// TIA Portal V20 program export: 7 tag tables, 9 data types, 119 data blocks, 46 code blocks (in call order from the OBs), 106 instance data blocks

VAR_GLOBAL   // PLC tag table "00_Simulation"
END_VAR

VAR_GLOBAL   // PLC tag table "06_ProductionData"
END_VAR
VAR_GLOBAL CONSTANT   // user constants
   NO_DATASETS_CYCLETIMER : Int := 14;   // SICAR: Number of data sets Cycle Timer
   NO_DATASETS_LIMITVALUES : Int := 2;   // SICAR: Number of data sets Limit Value
   NO_DATASETS_SHIFTCOUNTER : Int := 2;   // SICAR: Number of data sets Shift Counter
   NO_DATASETS_COUNTER : Int := 2;   // SICAR: Number of data sets Counter
END_VAR

VAR_GLOBAL   // PLC tag table "07_Energy"
   "Active energy export tariff 1(F)" AT %ID624 : Real;
   "Active energy import tariff 1(F)" AT %ID612 : Real;
   "Active power L1" AT %ID644 : Real;
   "Active power L2" AT %ID648 : Real;
   "Active power L3" AT %ID652 : Real;
   "Apparent energy tariff 1 (F)" AT %ID620 : Real;
   "Apparent power L1" AT %ID632 : Real;
   "Apparent power L2" AT %ID636 : Real;
   "Apparent power L3" AT %ID640 : Real;
   PAC3220InPut AT %I500.0 : "LER_typePAC3220Input_Status";
   "Reactive energy export tariff 1 (F)" AT %ID628 : Real;
   "Reactive energy import tariff 1 (F)" AT %ID616 : Real;
   "Reactive power L1" AT %ID656 : Real;
   "Reactive power L2" AT %ID660 : Real;
   "Reactive power L3" AT %ID664 : Real;
   PAC3220OutPut AT %Q500.0 : "LER_typePAC3220Output_Status";
END_VAR
VAR_GLOBAL CONSTANT   // user constants
   NO_OF_MACHINES : USInt := 1;   // SICAR: No of machines for EE-Monitor
   NO_OF_MEASUREPOINTS : USInt := 10;   // SICAR: No of measurepoints for EE-Monitor
   "DP_FRWA1_1_0_000CC1-KE50~DP_FRWA1_1_0_000CC1-KE50_900" : Hw_Io := 10;
END_VAR

VAR_GLOBAL   // PLC tag table "08_CmInfo"
END_VAR
VAR_GLOBAL CONSTANT   // user constants
   NO_OF_RF_IDENT_DEVICES : USInt := 1;   // SICAR: Number of RF readers
   NO_OF_MV_IDENT_DEVICES : USInt := 1;   // SICAR: Number of MV readers
   NO_OF_ET200SPMOTORSTARTER : USInt := 1;   // SICAR: Number of ET200SP Motorstarter
END_VAR

VAR_GLOBAL   // PLC tag table "11_Settings"
END_VAR
VAR_GLOBAL CONSTANT   // user constants
   MAX_NO_OF_DEVICES_X1 : Int := 200;
   MAX_NO_OF_MODULES_X1 : Int := 200;
   MAX_NO_OF_DEVICES_X2 : Int := 200;
   MAX_NO_OF_MODULES_X2 : Int := 200;
END_VAR

VAR_GLOBAL   // PLC tag table "CentralFunctions"
END_VAR

VAR_GLOBAL   // PLC tag table "TextListId"
END_VAR
VAR_GLOBAL CONSTANT   // user constants
   TEXT_LIST_ID_PN_DEV_DIAG : Int := 591;   // SICAR: ID of PLC Alarm text list
   TEXT_LIST_ID_CHECKSUM : Int := 584;   // SICAR: ID of PLC Alarm text list
   TEXT_LIST_ID_EEEMONITOR_REPORT : Int := 562;   // SICAR: ID of PLC Alarm text list
   TEXT_LIST_ID_EEEMONITOR_CALC : Int := 561;   // SICAR: ID of PLC Alarm text list
   TEXT_LIST_ID_IDENT_SYSTEM : Int := 516;   // SICAR: ID of PLC Alarm for ident demo
   TEXT_LIST_ID_SMC_PD : Int := 585;   // SICAR: ID of PLC Alarm text list
   TEXT_LIST_ID_MOTORSTARTERS : Int := 588;   // SICAR: ID of PLC Alarm for motorstarter Demo
   TEXT_LIST_ID_DEV_FWD_REV : Int := 592;   // SICAR: ID of PLC Alarm for motorstarter Demo
END_VAR

TYPE "typeInspectionToStack"
   STRUCT
      partOn : Bool;
      signal1 : Bool;
      signal2 : Bool;
      signal3 : Bool;
      signal4 : Bool;
      signal5 : Bool;
      signal6 : Bool;
      signal7 : Bool;
      signal8 : Bool;
      signal9 : Bool;
      signal10 : Bool;
      signal11 : Bool;
      signal12 : Bool;
      signal13 : Bool;
      signal14 : Bool;
      signal15 : Bool;
      readyForOperation : Bool;
      signal17 : Bool;
      signal18 : Bool;
      signal19 : Bool;
      signal20 : Bool;
      signal21 : Bool;
      signal22 : Bool;
      signal23 : Bool;
      signal24 : Bool;
      signal25 : Bool;
      signal26 : Bool;
      signal27 : Bool;
      signal28 : Bool;
      signal29 : Bool;
      signal30 : Bool;
      signal31 : Bool;
      noInterference : Bool;
      collisionAreaOn : Bool;
      collisionAreaOff : Bool;
      girpped : Bool;
      unGirpped : Bool;
      signal37 : Bool;
      signal38 : Bool;
      signal39 : Bool;
      signal40 : Bool;
      signal41 : Bool;
      signal42 : Bool;
      signal43 : Bool;
      signal44 : Bool;
      signal45 : Bool;
      signal46 : Bool;
      signal47 : Bool;
      loadEnable : Bool;
      unGripRequest : Bool;
      loadComplete : Bool;
      signal51 : Bool;
      signal52 : Bool;
      signal53 : Bool;
      signal54 : Bool;
      signal55 : Bool;
      signal56 : Bool;
      signal57 : Bool;
      signal58 : Bool;
      signal59 : Bool;
      signal60 : Bool;
      signal61 : Bool;
      signal62 : Bool;
      signal63 : Bool;
      signal64 : Bool;
      signal65 : Bool;
      signal66 : Bool;
      signal67 : Bool;
      signal68 : Bool;
      signal69 : Bool;
      signal70 : Bool;
      signal71 : Bool;
      signal72 : Bool;
      signal73 : Bool;
      signal74 : Bool;
      signal75 : Bool;
      signal76 : Bool;
      signal77 : Bool;
      signal78 : Bool;
      signal79 : Bool;
      signal80 : Bool;
      signal81 : Bool;
      signal82 : Bool;
      signal83 : Bool;
      signal84 : Bool;
      signal85 : Bool;
      signal86 : Bool;
      signal87 : Bool;
      signal88 : Bool;
      signal89 : Bool;
      signal90 : Bool;
      signal91 : Bool;
      signal92 : Bool;
      signal93 : Bool;
      signal94 : Bool;
      signal95 : Bool;
   END_STRUCT;
END_TYPE

TYPE "typeStackToInspection"
   STRUCT
      partOn : Bool;
      signal1 : Bool;
      signal2 : Bool;
      signal3 : Bool;
      signal4 : Bool;
      signal5 : Bool;
      signal6 : Bool;
      signal7 : Bool;
      signal8 : Bool;
      signal9 : Bool;
      signal10 : Bool;
      signal11 : Bool;
      signal12 : Bool;
      signal13 : Bool;
      signal14 : Bool;
      signal15 : Bool;
      readyForOperation : Bool;
      signal17 : Bool;
      signal18 : Bool;
      signal19 : Bool;
      signal20 : Bool;
      signal21 : Bool;
      signal22 : Bool;
      signal23 : Bool;
      signal24 : Bool;
      signal25 : Bool;
      signal26 : Bool;
      signal27 : Bool;
      signal28 : Bool;
      signal29 : Bool;
      signal30 : Bool;
      signal31 : Bool;
      noInterference : Bool;
      collisionAreaOn : Bool;
      collisionAreaOff : Bool;
      girpped : Bool;
      unGirpped : Bool;
      signal37 : Bool;
      signal38 : Bool;
      signal39 : Bool;
      signal40 : Bool;
      signal41 : Bool;
      signal42 : Bool;
      signal43 : Bool;
      signal44 : Bool;
      signal45 : Bool;
      signal46 : Bool;
      signal47 : Bool;
      unloadRequest : Bool;
      gripRequest : Bool;
      unLoadComplete : Bool;
      signal51 : Bool;
      signal52 : Bool;
      signal53 : Bool;
      signal54 : Bool;
      signal55 : Bool;
      signal56 : Bool;
      signal57 : Bool;
      signal58 : Bool;
      signal59 : Bool;
      signal60 : Bool;
      signal61 : Bool;
      signal62 : Bool;
      signal63 : Bool;
      signal64 : Bool;
      signal65 : Bool;
      signal66 : Bool;
      signal67 : Bool;
      signal68 : Bool;
      signal69 : Bool;
      signal70 : Bool;
      signal71 : Bool;
      signal72 : Bool;
      signal73 : Bool;
      signal74 : Bool;
      signal75 : Bool;
      signal76 : Bool;
      signal77 : Bool;
      signal78 : Bool;
      signal79 : Bool;
      signal80 : Bool;
      signal81 : Bool;
      signal82 : Bool;
      signal83 : Bool;
      signal84 : Bool;
      signal85 : Bool;
      signal86 : Bool;
      signal87 : Bool;
      signal88 : Bool;
      signal89 : Bool;
      signal90 : Bool;
      signal91 : Bool;
      signal92 : Bool;
      signal93 : Bool;
      signal94 : Bool;
      signal95 : Bool;
   END_STRUCT;
END_TYPE

TYPE "typeEmMotorStarterInterface"
// stored: Access Published
   STRUCT
      EMmotorstarter : Array[0.."NO_OF_EM"] of "typeMotorStarterInterface";
   END_STRUCT;
END_TYPE

TYPE "typeEt200SpMotorstarterInterfaceHmi"
// stored: Access Published
   STRUCT
      et200SpMotorstarterReadValue : Bool;   // read Value of MotorStarter
      et200SpNumberOfMotorstarters { ExternalWritable := 'False'} : USInt;   // Number of Motor Starters
      et200SpUnitMotorstarter : USInt := 1;   // Unit selected
      et200SpEMMotorstarter : USInt := 0;   // Equipment Module selected
      et200SpMotorstarterCurrent : Array[0.."NO_OF_ET200SPMOTORSTARTER"] of Real;   // Current values
      et200SpMotorstarterInputs : Array[0.."NO_OF_ET200SPMOTORSTARTER"] of "LSicar_typeMotorstarterIn";   // Motorstarter Data Inputs HMI
      et200SpMotorstarterOutputs : Array[0.."NO_OF_ET200SPMOTORSTARTER"] of "LSicar_typeMotorstarterOut";   // Motorstarter Data Outputs HMI
   END_STRUCT;
END_TYPE

TYPE "typeMotorStarterInterface"
// stored: Access Published
   STRUCT
      et200SpMotorstarterCurrent : Array[0.."NO_OF_ET200SPMOTORSTARTER"] of Real;   // Current values
      et200SpMotorstarterInputs : Array[0.."NO_OF_ET200SPMOTORSTARTER"] of "LSicar_typeMotorstarterIn";   // Motorstarter Data Inputs HMI
      et200SpMotorstarterOutputs : Array[0.."NO_OF_ET200SPMOTORSTARTER"] of "LSicar_typeMotorstarterOut";   // Motorstarter Data Outputs HMI
   END_STRUCT;
END_TYPE

TYPE "typeEMIdentMv"
// stored: Access Published
   STRUCT
      identMvEM : Array[0.."NO_OF_EM"] of "typeIdentMvHmi";
   END_STRUCT;
END_TYPE

TYPE "typeIdentMvHmi"
// stored: Access Published
   STRUCT
      selectedUnit : USInt;
      selectedEM : USInt;
      mvReaderId : USInt;   // MV Reader ID
      numberOfMv : USInt;   // Number of used MV readers
      mvReader : Array[0.."NO_OF_MV_IDENT_DEVICES"] of "LSicar_typeIdentInterfaceHmi";   // MV Reader
   END_STRUCT;
END_TYPE

TYPE "typeEMIdentRf"
// stored: Access Published
   STRUCT
      identRfEM : Array[0.."NO_OF_EM"] of "typeIdentRfHmi";
   END_STRUCT;
END_TYPE

TYPE "typeIdentRfHmi"
// stored: Access Published
   STRUCT
      selectedUnit : USInt;
      selectedEM : USInt;
      rfReaderId : USInt;   // RF Reader ID
      numberOfRf : USInt;   // Number of used RFIDs
      rfReader : Array[0.."NO_OF_RF_IDENT_DEVICES"] of "LSicar_typeIdentInterfaceHmi";   // RF Reader
   END_STRUCT;
END_TYPE

DATA_BLOCK "Hmi"   // DB199
// stored: MemoryReserve 100
   VAR
      mainHeader : Array[0.."NO_OF_PANELS"] of "LAF_typeHeader";   // Input from the status bar of the HMI
      operationInterlock : "LAF_typeOperationInterlockInterface";
   END_VAR
BEGIN
   mainHeader[0].plcToHmi.modeRequestsButtons.operatorControlAllowed := 16#003F;
   mainHeader[1].plcToHmi.stateCommandsButtons.visibility := 16#F;
   mainHeader[1].plcToHmi.stateCommandsButtons.operatorControlAllowed := 16#F;
   mainHeader[0].plcToHmi.specialFunctionButtons.visibility := 16#00330F7307337077;
   mainHeader[0].plcToHmi.specialFunctionButtons.operatorControlAllowed := 16#00330F7307337077;
END_DATA_BLOCK

DATA_BLOCK "LRemoteAccess_Data"   // DB275
TITLE = Data
AUTHOR : Siemens
// Storing data about mobile panel and UCP connection status
// stored: MemoryReserve 100
   VAR
      mobilePanel1 : "LRemoteAccess_typeMobilePanel";
      connectionBoxes : Array[1..2] of "LRemoteAccess_typeConnectionBox";
      ActivationMobileDP { S7_SetPoint := 'True'} : "LRemoteAccess_typeMobile_DeActivate";   // Activate Mobile Panel
      DeactivationMobileDP { S7_SetPoint := 'True'} : "LRemoteAccess_typeMobile_DeActivate";   // Deactivate Mobile Panel
      connectionTimeout { S7_SetPoint := 'True'} : Time := T#5s;   // Connection timeout. Keep greater than 3 sec. Default 5 sec.
   END_VAR
BEGIN
   connectionBoxes[1].ID := 20;
   connectionBoxes[2].ID := 21;
END_DATA_BLOCK

DATA_BLOCK "Simulation"   // DB134
TITLE = Simulation
// Simulation data
// stored: MemoryReserve 100
   VAR
      data : "LAF_typeSimulation";
   END_VAR
BEGIN
   data.simulationActiveHmi := true;
END_DATA_BLOCK

DATA_BLOCK "HMI_Interface_Overview"   // DB276
// stored: Access Published, MemoryReserve 100
   VAR
      State : Struct
         "Anode Reel Cut" : "HMI_IF_OverView_Unit_UDT";
         "Cathode Reel Cut" : "HMI_IF_OverView_Unit_UDT";
         "Stacker #1" : "HMI_IF_OverView_Unit_UDT";
         "Stacker #2" : "HMI_IF_OverView_Unit_UDT";
         Inspection : "HMI_IF_OverView_Unit_UDT";
      END_STRUCT;
      homeCodition : Array[0..13] of "LER_typeEmOverviewHomeCondition";
   END_VAR
BEGIN
END_DATA_BLOCK

DATA_BLOCK "HMI_Interface_Parameter"   // DB262
// stored: Access Published, MemoryReserve 100
   VAR
      ProcessUnitSelect : Int := 5;   // 1. Anode Reel Cut, 2. Cathode Reel Cut, 3. Stacking#1, 4.Stacking#2, 5. Inspection
      Recipe : "HMI_IF_Parameter_LIstRecipe_Interface";
   END_VAR
   VAR RETAIN
      Parameter : Array[0..20] of "HMI_IF_Parameter_Parameter_UDT";
      Softcam : Array[0..23] of "LER_typeSoftCamRelation";
   END_VAR
   VAR
      RecipeButton : "HMI_IF_Parameter_Save Button_UDT";
      FATModeSelect : "LER_TypeFATMode_ModeSelect";
   END_VAR
   VAR RETAIN
      FATModeInterface : "LER_TypeFATModeInterface";
   END_VAR
   VAR
      teachingPosInterface { S7_SetPoint := 'True'} : Array[0..48] of "LER_TypeTeachingPosInterface";
      TeachingPos_Index { S7_SetPoint := 'True'} : SInt;
   END_VAR
BEGIN
END_DATA_BLOCK

DATA_BLOCK "RecipeParameter"   // DB168
// stored: MemoryReserve 100
   VAR
      unitRecipe : "LER_typeRecipe";
      ParameterSV { S7_SetPoint := 'True'} : "HMI_IF_Parameter_ListRecipe_UDT";
      ParameterPV { S7_SetPoint := 'True'} : "HMI_IF_Parameter_ListRecipe_UDT";
   END_VAR
BEGIN
   ParameterSV.Recipe6 := 9000000.0;
   ParameterSV.Recipe7 := 9000000.0;
   ParameterPV.Recipe6 := 300000.0;
   ParameterPV.Recipe7 := 300000.0;
END_DATA_BLOCK

DATA_BLOCK "LAF_InternalManual"   // DB43
VERSION : 19.0
// stored: MemoryReserve 100
   VAR
      hmi : Array[1..1] of "LAF_typeManHmiDisp";   // number of HMIs - modify the array size based on the required HMIs
      manualOperationEnabled : Bool;   // feedback whether the manual operation lines are selected
      emsWithManualOpConfigured { ExternalWritable := 'False'} : "LGM_emsWithManualOpConfigured";   // List of EMs with manual operation configured, for HMI button visibility
      disableUnit1 { S7_SetPoint := 'True'} : Bool;
      RisingEdge : Bool;
   END_VAR
BEGIN
END_DATA_BLOCK

DATA_BLOCK "ManualOperationControl_Template"   // DB197
// stored: MemoryReserve 100
   VAR
      manualOperationEm { ExternalAccessible := 'False'; ExternalVisible := 'False'; ExternalWritable := 'False'} : "LAF_typeManEm";
      manualOperationEmArea { ExternalAccessible := 'False'; ExternalVisible := 'False'; ExternalWritable := 'False'} : Array[1..1] of "LAF_typeManOperationArea";
      manualOperationCms { ExternalAccessible := 'False'; ExternalVisible := 'False'; ExternalWritable := 'False'} : Array[1..1] of "LAF_typeManOperation";
   END_VAR
BEGIN
   manualOperationEm.equipmentModuleNum := 3400;
END_DATA_BLOCK

DATA_BLOCK "HMI_Interface_DeviceHistory"   // DB7
// stored: MemoryReserve 100
   VAR
      hotPressLeftHistory { ExternalWritable := 'False'; S7_SetPoint := 'True'} : "LER_typeVisionInspectData";
      hotPressRightHistory { ExternalWritable := 'False'; S7_SetPoint := 'True'} : "LER_typeVisionInspectData";
      hipotHistory { ExternalWritable := 'False'; S7_SetPoint := 'True'} : "LER_typeHipotDataLog";
      thicknessHistory { ExternalWritable := 'False'; S7_SetPoint := 'True'} : "LER_typeThicknessDataLog";
      visionHistory { ExternalWritable := 'False'; S7_SetPoint := 'True'} : "LER_typeVisionHistory";
      laserMarkHistory { ExternalWritable := 'False'; S7_SetPoint := 'True'} : "LER_typeQRMarkerDataLog";
      weightCheckHistory { ExternalWritable := 'False'; S7_SetPoint := 'True'} : "LER_typeWeightCheckDataLog";
   END_VAR
BEGIN
END_DATA_BLOCK

DATA_BLOCK "OperatorPrompts"   // DB123
// stored: Access Published, MemoryReserve 100
   VAR
      triggers { ExternalAccessible := 'False'; ExternalVisible := 'False'; ExternalWritable := 'False'} : Array[1..63] of Bool;
      activeOperatorPrompt { ExternalWritable := 'False'} : Int;
      ack : Bool;
   END_VAR
BEGIN
END_DATA_BLOCK

DATA_BLOCK "ProdDataInterfaceHmi"   // DB53
TITLE = HMI and user interface for production data
AUTHOR : SICAR
FAMILY : ProdData
// DESCRIPTION OF FUNCTIONS:
// stored: MemoryReserve 100
   VAR RETAIN
      numberOfDataSets : "LSicar_typeNumberOfDataSets";   // Number of configured data sets
   END_VAR
   VAR
      colorCodeLimitSummary : UInt;   // Overall status Limit values
      colorCodeLimitSelButton : Array[0..8] of UInt;   // Color code for data set select button (Limit values)
   END_VAR
   VAR RETAIN
      limitValueDataSetSel : Int := 1;   // selected data set limit values
      limitDataSet : Array[0.."NO_DATASETS_LIMITVALUES"] of "LSicar_typeLimitValue";   // Data sets limit .values
      cycleTimerDataSetSel : Int := 1;   // selected data set cycle timer
      cycleTimerDataSet : Array[0.."NO_DATASETS_CYCLETIMER"] of "LSicar_typeCycleTimer";   // Data sets cycle timer
      counterDataSetSel : Int := 1;   // selected data set counter
      counterDataSet : Array[0.."NO_DATASETS_COUNTER"] of "LSicar_typeCounter";   // Data sets counter
      shiftCounterDataSetSel : Int := 1;   // selected data set shift counter
      shiftCounterDataSet : Array[0.."NO_DATASETS_SHIFTCOUNTER"] of "LSicar_typeShiftCounter";   // Data sets shift counter
      shiftCountOeeDataSetSel : Int := 1;   // selected data set OEE
      shiftCounterOeeDataSet : Array[0.."NO_DATASETS_SHIFTCOUNTER"] of "LSicar_typeShiftCounterOee";   // Data sets shift counter OEE
   END_VAR
BEGIN
END_DATA_BLOCK

DATA_BLOCK "ProdDataSimulation"   // DB5
{ DB_Accessible_From_OPC_UA := 'FALSE' }
// stored: DBAccessibleFromOPCUA false, DBAccessibleFromWebserver false, MemoryReserve 100
   VAR
      ProdDataCounter { ExternalAccessible := 'False'; ExternalVisible := 'False'; ExternalWritable := 'False'} : Struct   // Test tag prod data
         ProdDataCounter1Up1 : Bool;   // Test tag prod data
         ProdDataCounter1Up2 : Bool;   // Test tag prod data
         ProdDataCounter1Down1 : Bool;   // Test tag prod data
         ProdDataCounter1Down2 : Bool;   // Test tag prod data
         ProdDataCounter1Reset1 : Bool;   // Test tag prod data
         ProdDataCounter1Reset2 : Bool;   // Test tag prod data
         ProdDataCounter1ResetAll : Bool;   // Test tag prod data
         ProdDataCounter2Up1 : Bool;
         ProdDataCounter2Up2 : Bool;
         ProdDataCounter2Down1 : Bool;
         ProdDataCounter2Down2 : Bool;
         ProdDataCounter2Reset1 : Bool;
         ProdDataCounter2Reset2 : Bool;
         ProdDataCounter2ResetAll : Bool;
         userInterfaceVisibilityDataSet2Counter : DWord := 2#0000_0000_0000_0000_0000_0000_0000_0011;
         userInterfaceVisibilityDataSet1Counter : DWord := 2#0000_0000_0000_0000_0011_1111_1111_1111;
         ProdDataEnable : Bool;
      END_STRUCT;
      ProdDataCyclic { ExternalAccessible := 'False'; ExternalVisible := 'False'; ExternalWritable := 'False'} : Struct   // Test tag prod data
         cycleTimer1Run1 : Bool;   // Test tag prod data
         cycleTimer1Run2 : Bool;   // Test tag prod data
         cycleTimer1Hold1 : Bool;   // Test tag prod data
         cycleTimer1Hold2 : Bool;   // Test tag prod data
         cycleTimer1Reset1 : Bool;   // Test tag prod data
         cycleTimer1Reset2 : Bool;   // Test tag prod data
         cycleTimer1ResetAll : Bool;   // Test tag prod data
         cycleTimer2Run1 : Bool;   // Test tag prod data
         cycleTimer2Run2 : Bool;   // Test tag prod data
         cycleTimer2Hold1 : Bool;   // Test tag prod data
         cycleTimer2Hold2 : Bool;   // Test tag prod data
         cycleTimer2Reset1 : Bool;   // Test tag prod data
         cycleTimer2Reset2 : Bool;   // Test tag prod data
         cycleTimer2ResetAll : Bool;   // Test tag prod data
         cyclicTimerEnable : Bool;
         userInterfaceVisibilityDataSet1Cyclic : DWord := 2#0000_0000_0000_0000_0000_0000_0000_0111;
         userInterfaceVisibilityDataSet2Cyclic : DWord := 2#0000_0000_0000_0000_0000_0000_0000_0111;
         userInterfaceVisibilityDataSet3Cyclic : DWord := 2#0000_0000_0000_0000_0000_0000_1110_1111;
         userInterfaceVisibilityDataSet4Cyclic : DWord := 2#0000_0000_0000_0000_0011_1110_1111_1011;
         userInterfaceVisibilityDataSet5Cyclic : DWord := 2#0000_0000_0000_1111_1110_1111_1111_0111;
         userInterfaceVisibilityDataSet6Cyclic : DWord := 2#0000_0000_0000_0111_1111_1101_1111_1111;
         userInterfaceVisibilityDataSet7Cyclic : DWord := 2#0000_0000_0000_0000_0000_0000_0000_1111;
         userInterfaceVisibilityDataSet8Cyclic : DWord := 2#0000_0000_0000_0000_0000_0000_0000_1111;
         userInterfaceVisibilityDataSet9Cyclic : DWord := 2#0000_0000_0000_0000_0000_0000_0000_1111;
         userInterfaceVisibilityDataSet10Cyclic : DWord := 2#0000_0000_0000_0000_0000_0000_0000_1111;
         userInterfaceVisibilityDataSet11Cyclic : DWord := 2#0000_0000_0000_0000_0000_0000_0000_1111;
         userInterfaceVisibilityDataSet12Cyclic : DWord := 2#0000_0000_0000_0000_0000_0000_0000_1111;
         userInterfaceVisibilityDataSet13Cyclic : DWord := 2#0000_0000_0000_0000_0000_0000_0000_0111;
         userInterfaceVisibilityDataSet14Cyclic : DWord := 2#0000_0000_0000_0000_0000_0000_0000_1111;
      END_STRUCT;
      ProdDataLimitValues { ExternalAccessible := 'False'; ExternalVisible := 'False'; ExternalWritable := 'False'} : Struct   // Test tag prod data
         limitVal1Count1PreWarn1 : Bool;   // Test tag prod data
         limitVal1Count1PreWarn3 : Bool;   // Test tag prod data
         limitVal1Count1PreWarn2 : Bool;   // Test tag prod data
         limitVal1Count1Alarm1 : Bool;   // Test tag prod data
         limitVal1Count1Alarm3 : Bool;   // Test tag prod data
         limitVal1Count1Alarm2 : Bool;   // Test tag prod data
         limitVal1Count1 : Bool;   // Test tag prod data
         limitVal1Count2 : Bool;   // Test tag prod data
         limitVal1Count3 : Bool;   // Test tag prod data
         limitVal1Set1 : Bool;   // Test tag prod data
         limitVal1Set3 : Bool;   // Test tag prod data
         limitVal1Set2 : Bool;   // Test tag prod data
         limitValuesEnable : Bool;
         userInterfaceVisibilityDataSet2LimitValues : DWord := 2#0000_0000_0000_0000_0000_0011_1111_1111;
         userInterfaceVisibilityDataSet1LimitValues : DWord := 2#0000_0000_0000_0000_0000_0000_0000_1111;
      END_STRUCT;
      ProdDataShiftCounter { ExternalAccessible := 'False'; ExternalVisible := 'False'; ExternalWritable := 'False'} : Struct   // Test tag prod data
         shiftCounter1Cnt1Curr : Bool;   // Test tag prod data
         shiftCounter1Cnt1CurrOk : Bool;   // Test tag prod data
         shiftCounter1Cnt2Curr : Bool;   // Test tag prod data
         shiftCounter1Cnt2CurrOk : Bool;   // Test tag prod data
         shiftCounter1Cnt3Curr : Bool;   // Test tag prod data
         shiftCounter1Cnt3CurrOk : Bool;   // Test tag prod data
         shiftCounter1ResetAllExt : Bool;   // Test tag prod data
         ShiftCounterEnable : Bool;
         userInterfaceVisibilityDataSet2ShiftCounter : DWord := 2#0000_0000_0000_0000_0000_0011_1111_1111;
         userInterfaceVisibilityDataSet1ShiftCounter : DWord := 2#0000_0000_0000_0000_0000_0000_0000_1111;
      END_STRUCT;
      ProdDataShiftCounterOEE { ExternalAccessible := 'False'; ExternalVisible := 'False'; ExternalWritable := 'False'} : Struct   // Test tag prod data
         ShiftCounterOEEEnable : Bool;
         userInterfaceVisibilityDataSet2ShiftCounterOEE : DWord := 2#0000_0000_0000_0000_0000_0011_1111_1111;
         userInterfaceVisibilityDataSet1ShiftCounterOEE : DWord := 2#0000_0000_0000_0000_0000_0000_0000_1111;
      END_STRUCT;
   END_VAR
BEGIN
END_DATA_BLOCK

DATA_BLOCK "ShiftInitBools"   // DB257
// stored: MemoryReserve 100
   VAR
      earlyShift : Bool;
      lateShift : Bool;
      nightShift : Bool;
   END_VAR
BEGIN
END_DATA_BLOCK

DATA_BLOCK "ShiftTimesList"   // DB52
TITLE = Shift times
{ DB_Accessible_From_OPC_UA := 'FALSE' }
AUTHOR : SICAR
FAMILY : Shiftmodel
// Shift times List
// stored: DBAccessibleFromOPCUA false, MemoryReserve 100
   VAR
      list { ExternalAccessible := 'False'; ExternalVisible := 'False'; ExternalWritable := 'False'} : Array[0..10] of "LSicar_typeShiftmodTime1DaySel";   // Shiftmodel list
   END_VAR
BEGIN
   list[3].listValidFor.sunday := TRUE;
   list[4].listValidFor.sunday := FALSE;
   list[1..3].listValidFor.monday := TRUE;
   list[4].listValidFor.monday := FALSE;
   list[1..3].listValidFor.tuesday := TRUE;
   list[4].listValidFor.tuesday := FALSE;
   list[1..3].listValidFor.wednesday := TRUE;
   list[4].listValidFor.wednesday := FALSE;
   list[1..3].listValidFor.thursday := TRUE;
   list[4].listValidFor.thursday := FALSE;
   list[1].listValidFor.friday := TRUE;
   list[3].listValidFor.friday := TRUE;
   list[4].listValidFor.friday := FALSE;
   list[3].listValidFor.saturday := TRUE;
   list[4].listValidFor.saturday := FALSE;
   list[1].shift[1].endCircuitTime := TOD#05:57:00;
   list[1].shift[2].endCircuitTime := TOD#13:57:00;
   list[1].shift[3].endCircuitTime := TOD#21:57:00;
   list[2].shift[1].endCircuitTime := TOD#04:57:00;
   list[2].shift[2].endCircuitTime := TOD#14:27:00;
   list[3].shift[1].endCircuitTime := TOD#05:57:00;
   list[3].shift[2].endCircuitTime := TOD#14:27:00;
   list[3].shift[3].endCircuitTime := TOD#22:57:00;
   list[4].shift[1..3].endCircuitTime := TOD#00:00:00;
   list[1].shift[1].start := TOD#06:00:00;
   list[1].shift[2].start := TOD#14:00:00;
   list[1].shift[3].start := TOD#22:00:00;
   list[2].shift[1].start := TOD#05:00:00;
   list[2].shift[2].start := TOD#14:30:00;
   list[3].shift[1].start := TOD#06:00:00;
   list[3].shift[2].start := TOD#14:30:00;
   list[3].shift[3].start := TOD#23:00:00;
   list[4].shift[1..3].start := TOD#00:00:00;
   list[1].shift[1].break[1].start := TOD#08:00:00;
   list[1].shift[1].break[2].start := TOD#10:00:00;
   list[1].shift[1].break[3].start := TOD#12:00:00;
   list[1].shift[1].break[4].start := TOD#00:00:00;
   list[1].shift[2].break[1].start := TOD#16:00:00;
   list[1].shift[2].break[2].start := TOD#18:00:00;
   list[1].shift[2].break[3].start := TOD#20:00:00;
   list[1].shift[3].break[1].start := TOD#00:00:00;
   list[1].shift[3].break[2].start := TOD#02:00:00;
   list[1].shift[3].break[3].start := TOD#04:00:00;
   list[2].shift[1].break[1].start := TOD#07:00:00;
   list[2].shift[1].break[2].start := TOD#09:00:00;
   list[2].shift[1].break[3].start := TOD#11:00:00;
   list[2].shift[1].break[4].start := TOD#13:00:00;
   list[2].shift[2].break[1].start := TOD#16:30:00;
   list[2].shift[2].break[2].start := TOD#18:30:00;
   list[2].shift[2].break[3].start := TOD#20:30:00;
   list[2].shift[2].break[4].start := TOD#22:00:00;
   list[3].shift[1].break[1].start := TOD#08:00:00;
   list[3].shift[1].break[2].start := TOD#10:00:00;
   list[3].shift[1].break[3].start := TOD#11:30:00;
   list[3].shift[1].break[4].start := TOD#12:30:00;
   list[3].shift[2].break[1].start := TOD#16:00:00;
   list[3].shift[2].break[2].start := TOD#18:00:00;
   list[3].shift[2].break[3].start := TOD#19:30:00;
   list[3].shift[2].break[4].start := TOD#20:30:00;
   list[3].shift[3].break[1].start := TOD#00:00:00;
   list[3].shift[3].break[2].start := TOD#02:00:00;
   list[3].shift[3].break[3].start := TOD#03:30:00;
   list[3].shift[3].break[4].start := TOD#04:30:00;
   list[4].shift[1].break[1..4].start := TOD#00:00:00;
   list[4].shift[2].break[1..4].start := TOD#00:00:00;
   list[4].shift[3].break[1..4].start := TOD#00:00:00;
   list[1].shift[1].break[1].startCircuitTime := TOD#08:02:00;
   list[1].shift[1].break[2].startCircuitTime := TOD#00:00:00;
   list[1].shift[1].break[3].startCircuitTime := TOD#12:02:00;
   list[1].shift[1].break[4].startCircuitTime := TOD#00:00:00;
   list[1].shift[2].break[1].startCircuitTime := TOD#16:02:00;
   list[1].shift[2].break[2].startCircuitTime := TOD#00:00:00;
   list[1].shift[2].break[3].startCircuitTime := TOD#20:02:00;
   list[1].shift[3].break[1].startCircuitTime := TOD#00:02:00;
   list[1].shift[3].break[2].startCircuitTime := TOD#00:00:00;
   list[1].shift[3].break[3].startCircuitTime := TOD#04:02:00;
   list[2].shift[1].break[1].startCircuitTime := TOD#07:02:00;
   list[2].shift[1].break[2].startCircuitTime := TOD#00:00:00;
   list[2].shift[1].break[3].startCircuitTime := TOD#11:02:00;
   list[2].shift[1].break[4].startCircuitTime := TOD#13:02:00;
   list[2].shift[2].break[1].startCircuitTime := TOD#16:32:00;
   list[2].shift[2].break[2].startCircuitTime := TOD#00:00:00;
   list[2].shift[2].break[3].startCircuitTime := TOD#20:32:00;
   list[2].shift[2].break[4].startCircuitTime := TOD#22:02:00;
   list[3].shift[1].break[1].startCircuitTime := TOD#00:00:00;
   list[3].shift[1].break[2].startCircuitTime := TOD#10:02:00;
   list[3].shift[1].break[3].startCircuitTime := TOD#00:00:00;
   list[3].shift[1].break[4].startCircuitTime := TOD#12:32:00;
   list[3].shift[2].break[1].startCircuitTime := TOD#00:00:00;
   list[3].shift[2].break[2].startCircuitTime := TOD#18:02:00;
   list[3].shift[2].break[3].startCircuitTime := TOD#00:00:00;
   list[3].shift[2].break[4].startCircuitTime := TOD#20:32:00;
   list[3].shift[3].break[1].startCircuitTime := TOD#00:00:00;
   list[3].shift[3].break[2].startCircuitTime := TOD#02:02:00;
   list[3].shift[3].break[3..4].startCircuitTime := TOD#00:00:00;
   list[4].shift[1].break[1..4].startCircuitTime := TOD#00:00:00;
   list[4].shift[2].break[1..4].startCircuitTime := TOD#00:00:00;
   list[4].shift[3].break[1..4].startCircuitTime := TOD#00:00:00;
   list[1].shift[1].break[1].endCircuitTime := TOD#08:13:00;
   list[1].shift[1].break[2].endCircuitTime := TOD#00:00:00;
   list[1].shift[1].break[3].endCircuitTime := TOD#12:13:00;
   list[1].shift[1].break[4].endCircuitTime := TOD#00:00:00;
   list[1].shift[2].break[1].endCircuitTime := TOD#16:13:00;
   list[1].shift[2].break[2].endCircuitTime := TOD#00:00:00;
   list[1].shift[2].break[3].endCircuitTime := TOD#20:13:00;
   list[1].shift[3].break[1].endCircuitTime := TOD#00:13:00;
   list[1].shift[3].break[2].endCircuitTime := TOD#00:00:00;
   list[1].shift[3].break[3].endCircuitTime := TOD#04:13:00;
   list[2].shift[1].break[1].endCircuitTime := TOD#07:13:00;
   list[2].shift[1].break[2].endCircuitTime := TOD#00:00:00;
   list[2].shift[1].break[3].endCircuitTime := TOD#11:13:00;
   list[2].shift[1].break[4].endCircuitTime := TOD#13:13:00;
   list[2].shift[2].break[1].endCircuitTime := TOD#16:43:00;
   list[2].shift[2].break[2].endCircuitTime := TOD#00:00:00;
   list[2].shift[2].break[3].endCircuitTime := TOD#20:43:00;
   list[2].shift[2].break[4].endCircuitTime := TOD#22:13:00;
   list[3].shift[1].break[1].endCircuitTime := TOD#00:00:00;
   list[3].shift[1].break[2].endCircuitTime := TOD#10:13:00;
   list[3].shift[1].break[3].endCircuitTime := TOD#00:00:00;
   list[3].shift[1].break[4].endCircuitTime := TOD#12:43:00;
   list[3].shift[2].break[1].endCircuitTime := TOD#00:00:00;
   list[3].shift[2].break[2].endCircuitTime := TOD#18:13:00;
   list[3].shift[2].break[3].endCircuitTime := TOD#00:00:00;
   list[3].shift[2].break[4].endCircuitTime := TOD#20:43:00;
   list[3].shift[3].break[1].endCircuitTime := TOD#00:00:00;
   list[3].shift[3].break[2].endCircuitTime := TOD#02:13:00;
   list[3].shift[3].break[3..4].endCircuitTime := TOD#00:00:00;
   list[4].shift[1].break[1..4].endCircuitTime := TOD#00:00:00;
   list[4].shift[2].break[1..4].endCircuitTime := TOD#00:00:00;
   list[4].shift[3].break[1..4].endCircuitTime := TOD#00:00:00;
   list[1].shift[1].break[1].end := TOD#08:15:00;
   list[1].shift[1].break[2].end := TOD#10:10:00;
   list[1].shift[1].break[3].end := TOD#12:15:00;
   list[1].shift[1].break[4].end := TOD#00:00:00;
   list[1].shift[2].break[1].end := TOD#16:15:00;
   list[1].shift[2].break[2].end := TOD#18:10:00;
   list[1].shift[2].break[3].end := TOD#20:15:00;
   list[1].shift[3].break[1].end := TOD#00:15:00;
   list[1].shift[3].break[2].end := TOD#02:10:00;
   list[1].shift[3].break[3].end := TOD#04:15:00;
   list[2].shift[1].break[1].end := TOD#07:15:00;
   list[2].shift[1].break[2].end := TOD#09:10:00;
   list[2].shift[1].break[3].end := TOD#11:15:00;
   list[2].shift[1].break[4].end := TOD#13:15:00;
   list[2].shift[2].break[1].end := TOD#16:45:00;
   list[2].shift[2].break[2].end := TOD#18:40:00;
   list[2].shift[2].break[3].end := TOD#20:45:00;
   list[2].shift[2].break[4].end := TOD#22:15:00;
   list[3].shift[1].break[1].end := TOD#08:10:00;
   list[3].shift[1].break[2].end := TOD#10:15:00;
   list[3].shift[1].break[3].end := TOD#11:40:00;
   list[3].shift[1].break[4].end := TOD#12:45:00;
   list[3].shift[2].break[1].end := TOD#16:10:00;
   list[3].shift[2].break[2].end := TOD#18:15:00;
   list[3].shift[2].break[3].end := TOD#19:40:00;
   list[3].shift[2].break[4].end := TOD#20:45:00;
   list[3].shift[3].break[1].end := TOD#00:10:00;
   list[3].shift[3].break[2].end := TOD#02:15:00;
   list[3].shift[3].break[3].end := TOD#03:40:00;
   list[3].shift[3].break[4].end := TOD#04:45:00;
   list[4].shift[1].break[1..4].end := TOD#00:00:00;
   list[4].shift[2].break[1..4].end := TOD#00:00:00;
   list[4].shift[3].break[1..4].end := TOD#00:00:00;
   list[1].shift[1].end := TOD#13:30:00;
   list[1].shift[2].end := TOD#21:30:00;
   list[1].shift[3].end := TOD#05:30:00;
   list[2].shift[1].end := TOD#14:00:00;
   list[2].shift[2].end := TOD#23:30:00;
   list[3].shift[1].end := TOD#13:30:00;
   list[3].shift[2].end := TOD#21:30:00;
   list[3].shift[3].end := TOD#05:30:00;
   list[4].shift[1..3].end := TOD#00:00:00;
   list[1].shift[1].startCircuitTime := TOD#13:33:00;
   list[1].shift[2].startCircuitTime := TOD#21:33:00;
   list[1].shift[3].startCircuitTime := TOD#05:33:00;
   list[2].shift[1].startCircuitTime := TOD#14:03:00;
   list[2].shift[2].startCircuitTime := TOD#23:33:00;
   list[3].shift[1].startCircuitTime := TOD#13:33:00;
   list[3].shift[2].startCircuitTime := TOD#21:33:00;
   list[3].shift[3].startCircuitTime := TOD#05:33:00;
   list[4].shift[1..3].startCircuitTime := TOD#00:00:00;
END_DATA_BLOCK

DATA_BLOCK "Settings"   // DB6
{ DB_Accessible_From_OPC_UA := 'FALSE' }
// stored: DBAccessibleFromOPCUA false, DBAccessibleFromWebserver false, MemoryReserve 100
   VAR
      diagPlc : "LAF_typePlcDiag";   // HMI interface PLC diag
      checksum : "LAF_typeChecksum";   // HMI interface PLCChecksum
      diagMemCard : "LAF_typeMemCardDiag";   // HMI interface SMCDiag
      cycleTimes : "LSicar_typeGlobalRuntime";
      setLocalPlcTime : "LAF_typeSetPlcTime";
      ITConnection : Bool := FALSE;   // Provides a visual representation of the connection with the IT systems.
   END_VAR
BEGIN
   diagPlc.im1PlantDesignLocIdent := 'GM BCDC';
   diagPlc.im1PlantDesignation := 'GM BCDC';
END_DATA_BLOCK

DATA_BLOCK "AxisConfigBackUp_DB"   // DB176
// stored: MemoryReserve 100
   VAR
      ManualSave : Bool;
   END_VAR
   VAR RETAIN
      DR1 : Struct
         cmJROutPnPLeftPositionX : Array[0..15] of "LBC_typeAxis64PosSetPosition";
      END_STRUCT;
      DR2 : Struct
         cmJROutPnPLeftPositionZ : Array[0..15] of "LBC_typeAxis64PosSetPosition";
      END_STRUCT;
      DR3 : Struct
         cmJROutPnPRightPositionX : Array[0..15] of "LBC_typeAxis64PosSetPosition";
      END_STRUCT;
      DR4 : Struct
         cmJROutPnPRightPositionZ : Array[0..15] of "LBC_typeAxis64PosSetPosition";
      END_STRUCT;
      DR5 : Struct
         cmTopTapingX : Array[0..15] of "LBC_typeAxis64PosSetPosition";
      END_STRUCT;
      DR6 : Struct
         cmTopTapingY : Array[0..15] of "LBC_typeAxis64PosSetPosition";
      END_STRUCT;
      DR7 : Struct
         cmJrFixStageX : Array[0..15] of "LBC_typeAxis64PosSetPosition";
      END_STRUCT;
      DR8 : Struct
         cmJrFixStageC : Array[0..15] of "LBC_typeAxis64PosSetPosition";
      END_STRUCT;
      DR9 : Struct
         cmSideTapingX : Array[0..15] of "LBC_typeAxis64PosSetPosition";
      END_STRUCT;
      DR10 : Struct
         cmSideTapingY : Array[0..15] of "LBC_typeAxis64PosSetPosition";
      END_STRUCT;
      DR11 : Struct
         cmHipotThicknessZ : Array[0..15] of "LBC_typeAxis64PosSetPosition";
      END_STRUCT;
      DR12 : Struct
         cmTransferPPLeftX : Array[0..15] of "LBC_typeAxis64PosSetPosition";
      END_STRUCT;
      DR13 : Struct
         cmTransferPPLeftY : Array[0..15] of "LBC_typeAxis64PosSetPosition";
      END_STRUCT;
      DR14 : Struct
         cmTransferPPLeftZ : Array[0..15] of "LBC_typeAxis64PosSetPosition";
      END_STRUCT;
      DR15 : Struct
         cmTransferPPRightX : Array[0..15] of "LBC_typeAxis64PosSetPosition";
      END_STRUCT;
      DR16 : Struct
         cmTransferPPRightY : Array[0..15] of "LBC_typeAxis64PosSetPosition";
      END_STRUCT;
      DR17 : Struct
         cmTransferPPRightZ : Array[0..15] of "LBC_typeAxis64PosSetPosition";
      END_STRUCT;
      DR18 : Struct
         cmJrUnloadingX : Array[0..15] of "LBC_typeAxis64PosSetPosition";
      END_STRUCT;
      DR19 : Struct
         cmJrUnloadingZ : Array[0..15] of "LBC_typeAxis64PosSetPosition";
      END_STRUCT;
      DR20 : Struct
         cmJrUnloadingC : Array[0..15] of "LBC_typeAxis64PosSetPosition";
      END_STRUCT;
   END_VAR
BEGIN
END_DATA_BLOCK

DATA_BLOCK "AxisDataBackUp_DB"   // DB137
// stored: Access Published, MemoryReserve 100
   VAR
      saveBit : Array[0..20] of Bool;   // DR save button
   END_VAR
   VAR RETAIN
      "emDistance[1]" { ExternalAccessible := 'False'; ExternalVisible := 'False'; ExternalWritable := 'False'} : "LER_typeDistanceInterface";
      "emDistance[2]" { ExternalAccessible := 'False'; ExternalVisible := 'False'; ExternalWritable := 'False'} : "LER_typeDistanceInterface";
      DR1 { ExternalAccessible := 'False'; ExternalVisible := 'False'; ExternalWritable := 'False'} : Struct
         "configuration.setPositions" : Array[0..15] of "LBC_typeAxis64PosSetPosition";
         softcam : "LER_typeSoftCamInterface";
      END_STRUCT;
      DR2 { ExternalAccessible := 'False'; ExternalVisible := 'False'; ExternalWritable := 'False'} : Struct
         "configuration.setPositions" : Array[0..15] of "LBC_typeAxis64PosSetPosition";
         softcam : "LER_typeSoftCamInterface";
      END_STRUCT;
      DR3 { ExternalAccessible := 'False'; ExternalVisible := 'False'; ExternalWritable := 'False'} : Struct
         "configuration.setPositions" : Array[0..15] of "LBC_typeAxis64PosSetPosition";
         softcam : "LER_typeSoftCamInterface";
      END_STRUCT;
      DR4 { ExternalAccessible := 'False'; ExternalVisible := 'False'; ExternalWritable := 'False'} : Struct
         "configuration.setPositions" : Array[0..15] of "LBC_typeAxis64PosSetPosition";
         softcam : "LER_typeSoftCamInterface";
      END_STRUCT;
      DR5 { ExternalAccessible := 'False'; ExternalVisible := 'False'; ExternalWritable := 'False'} : Struct
         "configuration.setPositions" : Array[0..15] of "LBC_typeAxis64PosSetPosition";
         softcam : "LER_typeSoftCamInterface";
      END_STRUCT;
      DR6 { ExternalAccessible := 'False'; ExternalVisible := 'False'; ExternalWritable := 'False'} : Struct
         "configuration.setPositions" : Array[0..15] of "LBC_typeAxis64PosSetPosition";
         softcam : "LER_typeSoftCamInterface";
      END_STRUCT;
      DR7 { ExternalAccessible := 'False'; ExternalVisible := 'False'; ExternalWritable := 'False'} : Struct
         "configuration.setPositions" : Array[0..15] of "LBC_typeAxis64PosSetPosition";
         softcam : "LER_typeSoftCamInterface";
      END_STRUCT;
      DR8 { ExternalAccessible := 'False'; ExternalVisible := 'False'; ExternalWritable := 'False'} : Struct
         "configuration.setPositions" : Array[0..15] of "LBC_typeAxis64PosSetPosition";
         softcam : "LER_typeSoftCamInterface";
      END_STRUCT;
      DR9 { ExternalAccessible := 'False'; ExternalVisible := 'False'; ExternalWritable := 'False'} : Struct
         "configuration.setPositions" : Array[0..15] of "LBC_typeAxis64PosSetPosition";
         softcam : "LER_typeSoftCamInterface";
      END_STRUCT;
      DR10 { ExternalAccessible := 'False'; ExternalVisible := 'False'; ExternalWritable := 'False'} : Struct
         "configuration.setPositions" : Array[0..15] of "LBC_typeAxis64PosSetPosition";
         softcam : "LER_typeSoftCamInterface";
      END_STRUCT;
      DR11 { ExternalAccessible := 'False'; ExternalVisible := 'False'; ExternalWritable := 'False'} : Struct
         "configuration.setPositions" : Array[0..15] of "LBC_typeAxis64PosSetPosition";
         softcam : "LER_typeSoftCamInterface";
      END_STRUCT;
      DR12 { ExternalAccessible := 'False'; ExternalVisible := 'False'; ExternalWritable := 'False'} : Struct
         "configuration.setPositions" : Array[0..15] of "LBC_typeAxis64PosSetPosition";
         softcam : "LER_typeSoftCamInterface";
      END_STRUCT;
      DR13 { ExternalAccessible := 'False'; ExternalVisible := 'False'; ExternalWritable := 'False'} : Struct
         "configuration.setPositions" : Array[0..15] of "LBC_typeAxis64PosSetPosition";
         softcam : "LER_typeSoftCamInterface";
      END_STRUCT;
      DR14 { ExternalAccessible := 'False'; ExternalVisible := 'False'; ExternalWritable := 'False'} : Struct
         "configuration.setPositions" : Array[0..15] of "LBC_typeAxis64PosSetPosition";
         softcam : "LER_typeSoftCamInterface";
      END_STRUCT;
      DR15 { ExternalAccessible := 'False'; ExternalVisible := 'False'; ExternalWritable := 'False'} : Struct
         "configuration.setPositions" : Array[0..15] of "LBC_typeAxis64PosSetPosition";
         softcam : "LER_typeSoftCamInterface";
      END_STRUCT;
      DR16 { ExternalAccessible := 'False'; ExternalVisible := 'False'; ExternalWritable := 'False'} : Struct
         "configuration.setPositions" : Array[0..15] of "LBC_typeAxis64PosSetPosition";
         softcam : "LER_typeSoftCamInterface";
      END_STRUCT;
      DR17 { ExternalAccessible := 'False'; ExternalVisible := 'False'; ExternalWritable := 'False'} : Struct
         "configuration.setPositions" : Array[0..15] of "LBC_typeAxis64PosSetPosition";
         softcam : "LER_typeSoftCamInterface";
      END_STRUCT;
      DR18 { ExternalAccessible := 'False'; ExternalVisible := 'False'; ExternalWritable := 'False'} : Struct
         "configuration.setPositions" : Array[0..15] of "LBC_typeAxis64PosSetPosition";
         softcam : "LER_typeSoftCamInterface";
      END_STRUCT;
      DR19 { ExternalAccessible := 'False'; ExternalVisible := 'False'; ExternalWritable := 'False'} : Struct
         "configuration.setPositions" : Array[0..15] of "LBC_typeAxis64PosSetPosition";
         softcam : "LER_typeSoftCamInterface";
      END_STRUCT;
      DR20 { ExternalAccessible := 'False'; ExternalVisible := 'False'; ExternalWritable := 'False'} : Struct
         "configuration.setPositions" : Array[0..15] of "LBC_typeAxis64PosSetPosition";
         softcam : "LER_typeSoftCamInterface";
      END_STRUCT;
   END_VAR
BEGIN
END_DATA_BLOCK

DATA_BLOCK "ManualOperationControl_U1Em0"   // DB104
// stored: MemoryReserve 100
   VAR
      manualOperationEm { ExternalAccessible := 'False'; ExternalVisible := 'False'; ExternalWritable := 'False'} : "LAF_typeManEm";
      manualOperationEmArea { ExternalAccessible := 'False'; ExternalVisible := 'False'; ExternalWritable := 'False'} : Array[1..2] of "LAF_typeManOperationArea";
      manualOperationCms { ExternalAccessible := 'False'; ExternalVisible := 'False'; ExternalWritable := 'False'} : Array[1..90] of "LAF_typeManOperation";
      axis { S7_SetPoint := 'True'} : Array[0..0] of "LBC_typeAxis64PosInterface";
      softCam { S7_SetPoint := 'True'} : Array[0..20] of "LER_typeSoftCamRelation";
      twoWayActuator { S7_SetPoint := 'True'} : Array[0..7] of "LBC_typeTwoWayActuatorInterface";
   END_VAR
BEGIN
   manualOperationEm.equipmentModuleNum := 1010;
   manualOperationEmArea[1].displayedLines := '1';
END_DATA_BLOCK

DATA_BLOCK "ManualOperationControl_U1Em1"   // DB21
// stored: MemoryReserve 100
   VAR
      manualOperationEm { ExternalAccessible := 'False'; ExternalVisible := 'False'; ExternalWritable := 'False'} : "LAF_typeManEm";
      manualOperationEmArea { ExternalAccessible := 'False'; ExternalVisible := 'False'; ExternalWritable := 'False'} : Array[1..2] of "LAF_typeManOperationArea";
      manualOperationCms { ExternalAccessible := 'False'; ExternalVisible := 'False'; ExternalWritable := 'False'} : Array[1..90] of "LAF_typeManOperation";
      axis { S7_SetPoint := 'True'} : Array[0..0] of "LBC_typeAxis64PosInterface";
      softCam { S7_SetPoint := 'True'} : Array[0..20] of "LER_typeSoftCamRelation";
      twoWayActuator { S7_SetPoint := 'True'} : Array[0..7] of "LBC_typeTwoWayActuatorInterface";
   END_VAR
BEGIN
   manualOperationEm.equipmentModuleNum := 1020;
   manualOperationEmArea[1].displayedLines := '1';
END_DATA_BLOCK

DATA_BLOCK "ManualOperationControl_U1Em10"   // DB28
// stored: MemoryReserve 100
   VAR
      manualOperationEm { ExternalAccessible := 'False'; ExternalVisible := 'False'; ExternalWritable := 'False'} : "LAF_typeManEm";
      manualOperationEmArea { ExternalAccessible := 'False'; ExternalVisible := 'False'; ExternalWritable := 'False'} : Array[1..2] of "LAF_typeManOperationArea";
      manualOperationCms { ExternalAccessible := 'False'; ExternalVisible := 'False'; ExternalWritable := 'False'} : Array[1..90] of "LAF_typeManOperation";
      axis { S7_SetPoint := 'True'} : Array[0..0] of "LBC_typeAxis64PosInterface";
      softCam { S7_SetPoint := 'True'} : Array[0..20] of "LER_typeSoftCamRelation";
      twoWayActuator { S7_SetPoint := 'True'} : Array[0..2] of "LBC_typeTwoWayActuatorInterface";
   END_VAR
BEGIN
   manualOperationEm.equipmentModuleNum := 1110;
   manualOperationEmArea[1].displayedLines := '1';
END_DATA_BLOCK

DATA_BLOCK "ManualOperationControl_U1Em11"   // DB24
// stored: MemoryReserve 100
   VAR
      manualOperationEm { ExternalAccessible := 'False'; ExternalVisible := 'False'; ExternalWritable := 'False'} : "LAF_typeManEm";
      manualOperationEmArea { ExternalAccessible := 'False'; ExternalVisible := 'False'; ExternalWritable := 'False'} : Array[1..2] of "LAF_typeManOperationArea";
      manualOperationCms { ExternalAccessible := 'False'; ExternalVisible := 'False'; ExternalWritable := 'False'} : Array[1..90] of "LAF_typeManOperation";
      axis { S7_SetPoint := 'True'} : Array[0..0] of "LBC_typeAxis64PosInterface";
      softCam { S7_SetPoint := 'True'} : Array[0..20] of "LER_typeSoftCamRelation";
      twoWayActuator { S7_SetPoint := 'True'} : Array[0..2] of "LBC_typeTwoWayActuatorInterface";
   END_VAR
BEGIN
   manualOperationEm.equipmentModuleNum := 1120;
   manualOperationEmArea[1].displayedLines := '1';
END_DATA_BLOCK

DATA_BLOCK "ManualOperationControl_U1Em12"   // DB33
// stored: MemoryReserve 100
   VAR
      manualOperationEm { ExternalAccessible := 'False'; ExternalVisible := 'False'; ExternalWritable := 'False'} : "LAF_typeManEm";
      manualOperationEmArea { ExternalAccessible := 'False'; ExternalVisible := 'False'; ExternalWritable := 'False'} : Array[1..2] of "LAF_typeManOperationArea";
      manualOperationCms { ExternalAccessible := 'False'; ExternalVisible := 'False'; ExternalWritable := 'False'} : Array[1..90] of "LAF_typeManOperation";
      axis { S7_SetPoint := 'True'} : Array[0..0] of "LBC_typeAxis64PosInterface";
      softCam { S7_SetPoint := 'True'} : Array[0..20] of "LER_typeSoftCamRelation";
      twoWayActuator { S7_SetPoint := 'True'} : Array[0..7] of "LBC_typeTwoWayActuatorInterface";
   END_VAR
BEGIN
   manualOperationEm.equipmentModuleNum := 1130;
   manualOperationEmArea[1].displayedLines := '1';
END_DATA_BLOCK

DATA_BLOCK "ManualOperationControl_U1Em13"   // DB17
// stored: MemoryReserve 100
   VAR
      manualOperationEm { ExternalAccessible := 'False'; ExternalVisible := 'False'; ExternalWritable := 'False'} : "LAF_typeManEm";
      manualOperationEmArea { ExternalAccessible := 'False'; ExternalVisible := 'False'; ExternalWritable := 'False'} : Array[1..2] of "LAF_typeManOperationArea";
      manualOperationCms { ExternalAccessible := 'False'; ExternalVisible := 'False'; ExternalWritable := 'False'} : Array[1..90] of "LAF_typeManOperation";
      axis { S7_SetPoint := 'True'} : Array[0..3] of "LBC_typeAxis64PosInterface";
      softCam { S7_SetPoint := 'True'} : Array[0..20] of "LER_typeSoftCamRelation";
      twoWayActuator { S7_SetPoint := 'True'} : Array[0..1] of "LBC_typeTwoWayActuatorInterface";
   END_VAR
BEGIN
   manualOperationEm.equipmentModuleNum := 1140;
   manualOperationEmArea[1].displayedLines := '1';
END_DATA_BLOCK

DATA_BLOCK "ManualOperationControl_U1Em14"   // DB13
// stored: MemoryReserve 100
   VAR
      manualOperationEm { ExternalAccessible := 'False'; ExternalVisible := 'False'; ExternalWritable := 'False'} : "LAF_typeManEm";
      manualOperationEmArea { ExternalAccessible := 'False'; ExternalVisible := 'False'; ExternalWritable := 'False'} : Array[1..2] of "LAF_typeManOperationArea";
      manualOperationCms { ExternalAccessible := 'False'; ExternalVisible := 'False'; ExternalWritable := 'False'} : Array[1..90] of "LAF_typeManOperation";
      axis { S7_SetPoint := 'True'} : Array[0..0] of "LBC_typeAxis64PosInterface";
      softCam { S7_SetPoint := 'True'} : Array[0..0] of "LER_typeSoftCamInterface";
      twoWayActuator { S7_SetPoint := 'True'} : Array[0..0] of "LBC_typeTwoWayActuatorInterface";
   END_VAR
BEGIN
   manualOperationEm.equipmentModuleNum := 1150;
   manualOperationEmArea[1].displayedLines := '1';
END_DATA_BLOCK

DATA_BLOCK "ManualOperationControl_U1Em15"   // DB75
// stored: MemoryReserve 100
   VAR
      manualOperationEm { ExternalAccessible := 'False'; ExternalVisible := 'False'; ExternalWritable := 'False'} : "LAF_typeManEm";
      manualOperationEmArea { ExternalAccessible := 'False'; ExternalVisible := 'False'; ExternalWritable := 'False'} : Array[1..2] of "LAF_typeManOperationArea";
      manualOperationCms { ExternalAccessible := 'False'; ExternalVisible := 'False'; ExternalWritable := 'False'} : Array[1..90] of "LAF_typeManOperation";
      axis { S7_SetPoint := 'True'} : Array[0..0] of "LBC_typeAxis64PosInterface";
      softCam { S7_SetPoint := 'True'} : Array[0..0] of "LER_typeSoftCamInterface";
      twoWayActuator : Array[0..0] of "LBC_typeTwoWayActuatorInterface";
   END_VAR
BEGIN
   manualOperationEm.equipmentModuleNum := 1160;
   manualOperationEmArea[1].displayedLines := '1';
END_DATA_BLOCK

DATA_BLOCK "ManualOperationControl_U1Em2"   // DB57
// stored: MemoryReserve 100
   VAR
      manualOperationEm { ExternalAccessible := 'False'; ExternalVisible := 'False'; ExternalWritable := 'False'} : "LAF_typeManEm";
      manualOperationEmArea { ExternalAccessible := 'False'; ExternalVisible := 'False'; ExternalWritable := 'False'} : Array[1..2] of "LAF_typeManOperationArea";
      manualOperationCms { ExternalAccessible := 'False'; ExternalVisible := 'False'; ExternalWritable := 'False'} : Array[1..90] of "LAF_typeManOperation";
      axis { S7_SetPoint := 'True'} : Array[0..4] of "LBC_typeAxis64PosInterface";
      softCam { S7_SetPoint := 'True'} : Array[0..20] of "LER_typeSoftCamRelation";
      twoWayActuator { S7_SetPoint := 'True'} : Array[0..2] of "LBC_typeTwoWayActuatorInterface";
   END_VAR
BEGIN
   manualOperationEm.equipmentModuleNum := 1030;
   manualOperationEmArea[1].displayedLines := '1';
END_DATA_BLOCK

DATA_BLOCK "ManualOperationControl_U1Em3"   // DB107
// stored: MemoryReserve 100
   VAR
      manualOperationEm { ExternalAccessible := 'False'; ExternalVisible := 'False'; ExternalWritable := 'False'} : "LAF_typeManEm";
      manualOperationEmArea { ExternalAccessible := 'False'; ExternalVisible := 'False'; ExternalWritable := 'False'} : Array[1..2] of "LAF_typeManOperationArea";
      manualOperationCms { ExternalAccessible := 'False'; ExternalVisible := 'False'; ExternalWritable := 'False'} : Array[1..90] of "LAF_typeManOperation";
      axis { S7_SetPoint := 'True'} : Array[0..2] of "LBC_typeAxis64PosInterface";
      softCam { S7_SetPoint := 'True'} : Array[0..20] of "LER_typeSoftCamRelation";
      twoWayActuator { S7_SetPoint := 'True'} : Array[0..11] of "LBC_typeTwoWayActuatorInterface";
   END_VAR
BEGIN
   manualOperationEm.equipmentModuleNum := 1040;
END_DATA_BLOCK

DATA_BLOCK "ManualOperationControl_U1Em4"   // DB26
// stored: MemoryReserve 100
   VAR
      manualOperationEm { ExternalAccessible := 'False'; ExternalVisible := 'False'; ExternalWritable := 'False'} : "LAF_typeManEm";
      manualOperationEmArea { ExternalAccessible := 'False'; ExternalVisible := 'False'; ExternalWritable := 'False'} : Array[1..2] of "LAF_typeManOperationArea";
      manualOperationCms { ExternalAccessible := 'False'; ExternalVisible := 'False'; ExternalWritable := 'False'} : Array[1..90] of "LAF_typeManOperation";
      axis { S7_SetPoint := 'True'} : Array[0..4] of "LBC_typeAxis64PosInterface";
      softCam { S7_SetPoint := 'True'} : Array[0..20] of "LER_typeSoftCamRelation";
      twoWayActuator { S7_SetPoint := 'True'} : Array[0..13] of "LBC_typeTwoWayActuatorInterface";
   END_VAR
BEGIN
   manualOperationEm.equipmentModuleNum := 1050;
   manualOperationEmArea[1].displayedLines := '1';
END_DATA_BLOCK

DATA_BLOCK "ManualOperationControl_U1Em5"   // DB22
// stored: MemoryReserve 100
   VAR
      manualOperationEm { ExternalAccessible := 'False'; ExternalVisible := 'False'; ExternalWritable := 'False'} : "LAF_typeManEm";
      manualOperationEmArea { ExternalAccessible := 'False'; ExternalVisible := 'False'; ExternalWritable := 'False'} : Array[1..2] of "LAF_typeManOperationArea";
      manualOperationCms { ExternalAccessible := 'False'; ExternalVisible := 'False'; ExternalWritable := 'False'} : Array[1..90] of "LAF_typeManOperation";
      axis { S7_SetPoint := 'True'} : Array[0..6] of "LBC_typeAxis64PosInterface";
      softCam { S7_SetPoint := 'True'} : Array[0..20] of "LER_typeSoftCamRelation";
      twoWayActuator { S7_SetPoint := 'True'} : Array[0..2] of "LBC_typeTwoWayActuatorInterface";
   END_VAR
BEGIN
   manualOperationEm.equipmentModuleNum := 1060;
   manualOperationEmArea[1].displayedLines := '1';
END_DATA_BLOCK

DATA_BLOCK "ManualOperationControl_U1Em6"   // DB25
// stored: MemoryReserve 100
   VAR
      manualOperationEm { ExternalAccessible := 'False'; ExternalVisible := 'False'; ExternalWritable := 'False'} : "LAF_typeManEm";
      manualOperationEmArea { ExternalAccessible := 'False'; ExternalVisible := 'False'; ExternalWritable := 'False'} : Array[1..2] of "LAF_typeManOperationArea";
      manualOperationCms { ExternalAccessible := 'False'; ExternalVisible := 'False'; ExternalWritable := 'False'} : Array[1..90] of "LAF_typeManOperation";
      axis { S7_SetPoint := 'True'} : Array[0..0] of "LBC_typeAxis64PosInterface";
      softCam { S7_SetPoint := 'True'} : Array[0..20] of "LER_typeSoftCamRelation";
      twoWayActuator { S7_SetPoint := 'True'} : Array[0..4] of "LBC_typeTwoWayActuatorInterface";
   END_VAR
BEGIN
   manualOperationEm.equipmentModuleNum := 1070;
   manualOperationEmArea[1].displayedLines := '1';
END_DATA_BLOCK

DATA_BLOCK "ManualOperationControl_U1Em7"   // DB27
// stored: MemoryReserve 100
   VAR
      manualOperationEm { ExternalAccessible := 'False'; ExternalVisible := 'False'; ExternalWritable := 'False'} : "LAF_typeManEm";
      manualOperationEmArea { ExternalAccessible := 'False'; ExternalVisible := 'False'; ExternalWritable := 'False'} : Array[1..2] of "LAF_typeManOperationArea";
      manualOperationCms { ExternalAccessible := 'False'; ExternalVisible := 'False'; ExternalWritable := 'False'} : Array[1..90] of "LAF_typeManOperation";
      axis { S7_SetPoint := 'True'} : Array[0..0] of "LBC_typeAxis64PosInterface";
      softCam { S7_SetPoint := 'True'} : Array[0..20] of "LER_typeSoftCamRelation";
      twoWayActuator { S7_SetPoint := 'True'} : Array[0..4] of "LBC_typeTwoWayActuatorInterface";
   END_VAR
BEGIN
   manualOperationEm.equipmentModuleNum := 1080;
   manualOperationEmArea[1].displayedLines := '1';
END_DATA_BLOCK

DATA_BLOCK "ManualOperationControl_U1Em8"   // DB35
// stored: MemoryReserve 100
   VAR
      manualOperationEm { ExternalAccessible := 'False'; ExternalVisible := 'False'; ExternalWritable := 'False'} : "LAF_typeManEm";
      manualOperationEmArea { ExternalAccessible := 'False'; ExternalVisible := 'False'; ExternalWritable := 'False'} : Array[1..2] of "LAF_typeManOperationArea";
      manualOperationCms { ExternalAccessible := 'False'; ExternalVisible := 'False'; ExternalWritable := 'False'} : Array[1..40] of "LAF_typeManOperation";
      axis { S7_SetPoint := 'True'} : Array[0..1] of "LBC_typeAxis64PosInterface";
      softCam { S7_SetPoint := 'True'} : Array[0..20] of "LER_typeSoftCamRelation";
      twoWayActuator { S7_SetPoint := 'True'} : Array[0..7] of "LBC_typeTwoWayActuatorInterface";
   END_VAR
BEGIN
   manualOperationEm.equipmentModuleNum := 1090;
   manualOperationEmArea[1].displayedLines := '1';
END_DATA_BLOCK

DATA_BLOCK "ManualOperationControl_U1Em9"   // DB14
// stored: MemoryReserve 100
   VAR
      manualOperationEm { ExternalAccessible := 'False'; ExternalVisible := 'False'; ExternalWritable := 'False'} : "LAF_typeManEm";
      manualOperationEmArea { ExternalAccessible := 'False'; ExternalVisible := 'False'; ExternalWritable := 'False'} : Array[1..2] of "LAF_typeManOperationArea";
      manualOperationCms { ExternalAccessible := 'False'; ExternalVisible := 'False'; ExternalWritable := 'False'} : Array[1..90] of "LAF_typeManOperation";
      axis { S7_SetPoint := 'True'} : Array[0..0] of "LBC_typeAxis64PosInterface";
      softCam { S7_SetPoint := 'True'} : Array[0..20] of "LER_typeSoftCamRelation";
      twoWayActuator { S7_SetPoint := 'True'} : Array[0..2] of "LBC_typeTwoWayActuatorInterface";
   END_VAR
BEGIN
   manualOperationEm.equipmentModuleNum := 1100;
   manualOperationEmArea[1].displayedLines := '1';
END_DATA_BLOCK

DATA_BLOCK "DriveDiagConfig"   // DB12
TITLE = DriveDiagConfig
AUTHOR : Siemens Digital Industries
FAMILY : LAF
NAME : LAF_DriveDiagConfigData
VERSION : 1.1
// Configuration data array for drive diagnostic
// stored: MemoryReserve 100
   VAR
      driveObjects : Array[0.."LAF_DRV_DIAG_NO_DO"] of "LAF_typeDriveDiagConfig";
      torqueLoad : Array[0.."LAF_DRV_DIAG_NO_DO"] of "LER_typeServoTorqueCalConfigruation";
   END_VAR
BEGIN
END_DATA_BLOCK

DATA_BLOCK "DriveDiagInterfaceHmi"   // DB46
TITLE = DriveDiagInterfaceHmi
AUTHOR : Siemens Digital Industries
FAMILY : LAF
NAME : LAF_DriveDiagInterfaceHmi
VERSION : 1.1
// HMI interface for drive diagnostic
// stored: MemoryReserve 100
   VAR
      diagStatus : "LAF_typeDriveDiagInterfaceHmi";
      torqueLoad : Array[0.."LAF_DRV_DIAG_NO_DO"] of "LER_typeServoTorqueCalInterface";
   END_VAR
BEGIN
END_DATA_BLOCK

DATA_BLOCK "IdentData"   // DB221
TITLE = Interface read/write data
AUTHOR : SICAR
FAMILY : Ident
VERSION : 1.0
// Ident data
// stored: MemoryReserve 100
   VAR
      rfReader { ExternalAccessible := 'False'; ExternalVisible := 'False'; ExternalWritable := 'False'} : Array[0.."NO_OF_RF_IDENT_DEVICES"] of "LSicar_typeIdentReadWriteDat";   // Reader
      mvReader { S7_SetPoint := 'True'} : Array[0.."NO_OF_MV_IDENT_DEVICES"] of "LSicar_typeIdentReadWriteDat";
   END_VAR
BEGIN
END_DATA_BLOCK

DATA_BLOCK "TestVarIdent"   // DB76
TITLE = Test tags for ident
AUTHOR : SICAR
FAMILY : Ident
VERSION : 1.0
// Test tags for ident
// stored: MemoryReserve 100
   VAR
      init1 : Bool;   // Init 1
      read1 : Bool;   // Read1
      write1 : Bool;   // Write1
      init2 : Bool;   // Init 2
      read2 : Bool;   // Read2
      write2 : Bool;   // Write2
      testString : String[32];   // Test string
      charArr : Array[1..32] of Byte;   // Character Array
      prgNoMan : USInt;   // Program number manual
      enableManCtrlRf : Bool := false;   // Enable manual control RFID
      enableOption : Bool;   // Enable options
      enableManCtrlMV : Bool;   // Enable manual control MV
   END_VAR
BEGIN
END_DATA_BLOCK

DATA_BLOCK "InterfaceSignals"   // DB196
// stored: MemoryReserve 100
   VAR
      HMI_Interface_Mode : Bool;
      "Button Value" : Array[0..99] of "LER_SignalsInput";
   END_VAR
BEGIN
END_DATA_BLOCK

DATA_BLOCK "TestVarMortorstarter"   // DB223
// stored: MemoryReserve 100
   VAR
      TestplantIdentifier : WString[24] := WSTRING#'++0.000MS1';
      faceplateType : USInt;   // Bit for showing the buttons on FP
      operatorTripReset : Bool;   // Operator Trip Reset Motorstarter
      contactorControlOn { S7_SetPoint := 'True'} : Bool;
   END_VAR
BEGIN
END_DATA_BLOCK

DATA_BLOCK "OtherSafetyInterface"   // DB211
// stored: MemoryReserve 100
   VAR
      OtherDoor1 : "LER_typefDoorInterface";   // BA010 Other Door
      OtherDoor2 : "LER_typefDoorInterface";   // BA015 Other Door
      OtherDoor3 : "LER_typefDoorInterface";   // BA030 Other Door
      OtherDoor4 : "LER_typefDoorInterface";   // BA040 Other Door
      InspectionExternalDoor { S7_SetPoint := 'True'} : "LER_typefDoorInterface";   // Inspection External Door
      Inspection30MaintDoor { S7_SetPoint := 'True'} : "LER_typefDoorInterface";   // Inspection BA030 Main Door
      Inspection40MaintDoor { S7_SetPoint := 'True'} : "LER_typefDoorInterface";   // Inspection BA040 Main Door
      OtherEMO1 { S7_SetPoint := 'True'} : Bool;   // BA010 EMO
      OtherEMO2 { S7_SetPoint := 'True'} : Bool;   // BA015 EMO
      OtherEMO3 { S7_SetPoint := 'True'} : Bool;   // BA030 EMO
      OtherEMO4 { S7_SetPoint := 'True'} : Bool;   // BA040 EMO
      Inspection30LightCurtain { S7_SetPoint := 'True'} : "LER_typeLightCurtainInterface";   // BA060 Stack #1 Light Curatain
      Inspection40LightCurtain { S7_SetPoint := 'True'} : "LER_typeLightCurtainInterface";   // BA060 Stack #2 Light Curatain
      "30CathodeConveyorCover" { S7_SetPoint := 'True'} : "LER_typeConveyorCoverInterface";   // BA030 Cathode Conveyor Cover
      "30AnodeConveyorCover" { S7_SetPoint := 'True'} : "LER_typeConveyorCoverInterface";   // BA030 Cathode Anode Cover
      "40CathodeConveyorCover" { S7_SetPoint := 'True'} : "LER_typeConveyorCoverInterface";   // BA040 Cathode Conveyor Cover
      "40AnodeConveyorCover" { S7_SetPoint := 'True'} : "LER_typeConveyorCoverInterface";   // BA040 Cathode Anode Cover
   END_VAR
BEGIN
   OtherDoor1.configuration.referenceDesignator := WSTRING#'BA010';
   OtherDoor2.configuration.referenceDesignator := WSTRING#'BA015';
   OtherDoor3.configuration.referenceDesignator := WSTRING#'BA030';
   OtherDoor4.configuration.referenceDesignator := WSTRING#'BA040';
   InspectionExternalDoor.configuration.referenceDesignator := WSTRING#'External';
   Inspection30MaintDoor.configuration.referenceDesignator := WSTRING#'30';
   Inspection40MaintDoor.configuration.referenceDesignator := WSTRING#'40';
   Inspection30LightCurtain.configuration.referenceDesignator := WSTRING#'STK1';
   Inspection40LightCurtain.configuration.referenceDesignator := WSTRING#'STK2';
   "30CathodeConveyorCover".configuration.referenceDesignator := WSTRING#'30Cath';
   "30AnodeConveyorCover".configuration.referenceDesignator := WSTRING#'30Anod';
   "40CathodeConveyorCover".configuration.referenceDesignator := WSTRING#'40Cath';
   "40AnodeConveyorCover".configuration.referenceDesignator := WSTRING#'40Anod';
END_DATA_BLOCK

DATA_BLOCK "SafetyDoorInterface"   // DB179
// stored: Access Published, MemoryReserve 100
   VAR
      fDoor11Interface { S7_SetPoint := 'True'} : "LER_typefDoorInterface";
      fDoor10Interface { S7_SetPoint := 'True'} : "LER_typefDoorInterface";
      fDoor9Interface { S7_SetPoint := 'True'} : "LER_typefDoorInterface";
      fDoor8Interface { S7_SetPoint := 'True'} : "LER_typefDoorInterface";
      fDoor7Interface { S7_SetPoint := 'True'} : "LER_typefDoorInterface";
      fDoor6Interface { S7_SetPoint := 'True'} : "LER_typefDoorInterface";
      fDoor5Interface { S7_SetPoint := 'True'} : "LER_typefDoorInterface";
      fDoor4Interface { S7_SetPoint := 'True'} : "LER_typefDoorInterface";
      fDoor3Interface { S7_SetPoint := 'True'} : "LER_typefDoorInterface";
      fDoor2Interface { S7_SetPoint := 'True'} : "LER_typefDoorInterface";
      fDoor1Interface { S7_SetPoint := 'True'} : "LER_typefDoorInterface";
      TON { S7_SetPoint := 'True'} : Array[0..9] of TON_TIME;
   END_VAR
BEGIN
   fDoor11Interface.configuration.referenceDesignator := WSTRING#'MAINT';
   fDoor10Interface.configuration.referenceDesignator := WSTRING#'STK1';
   fDoor9Interface.configuration.referenceDesignator := WSTRING#'STK2';
   fDoor8Interface.configuration.referenceDesignator := WSTRING#'TR.PP L';
   fDoor7Interface.configuration.referenceDesignator := WSTRING#'TR.PP';
   fDoor6Interface.configuration.referenceDesignator := WSTRING#'UNLOAD';
   fDoor5Interface.configuration.referenceDesignator := WSTRING#'WEIGHT';
   fDoor4Interface.configuration.referenceDesignator := WSTRING#'LASER';
   fDoor3Interface.configuration.referenceDesignator := WSTRING#'H.PRESS';
   fDoor2Interface.configuration.referenceDesignator := WSTRING#'S.TAPE';
   fDoor1Interface.configuration.referenceDesignator := WSTRING#'T.TAPE';
END_DATA_BLOCK

DATA_BLOCK "E2MSimulation"   // DB23
{ DB_Accessible_From_OPC_UA := 'FALSE' }
// stored: DBAccessibleFromOPCUA false, DBAccessibleFromWebserver false, MemoryReserve 100
   VAR
      randomNumber : Real;   // Randomly generated number
   END_VAR
BEGIN
END_DATA_BLOCK

DATA_BLOCK "BK01"   // DB298
// stored: Access Published, MemoryReserve 100
   VAR
      "X10-1 JR OUT P&P1 Y-AXIS ROBOT LIMIT SENSOR(-)" : Bool;
      "X11-1 JR OUT P&P1 Y-AXIS ROBOT LIMIT SENSOR(+)" : Bool;
      "X12-1 JR OUT P&P2 Y-AXIS ROBOT LIMIT SENSOR(-)" : Bool;
      "X13-1 JR OUT P&P2 Y-AXIS ROBOT LIMIT SENSOR(+)" : Bool;
      "X14-1 STACK 1 NG BOX DETECT SENSOR" : Bool;
      "X15-1 SPARE" : Bool;
      "X16-1 SPARE" : Bool;
      "X17-1 SPARE" : Bool;
      "X10-2 JR OUT P&P1 Y-AXIS ROBOT HOME SENSOR" : Bool;
      "X11-2 SPARE" : Bool;
      "X12-2 JR OUT P&P2 Y-AXIS ROBOT HOME SENSOR" : Bool;
      "X13-2 SPARE" : Bool;
      "X14-2 STACK 2 NG BOX DETECT SENSOR" : Bool;
      "X15-2 SPARE" : Bool;
      "X16-2 SPARE" : Bool;
      "X17-2 SPARE" : Bool;
   END_VAR
BEGIN
END_DATA_BLOCK

DATA_BLOCK "BK02"   // DB299
// stored: MemoryReserve 100
   VAR
      "X10-1 JR OUT P&P1 Z-AXIS LIMIT SENSOR(-)" : Bool;
      "X10-2 JR OUT P&P1 Z-AXIS HOME SENSOR" : Bool;
      "X12-1 JR OUT P&P1 Z-AXIS LIMIT SENSOR(+)" : Bool;
      "X12-2 JR OUT P&P1 STACK DETECT SENSOR" : Bool;
      "X14-1 JR OUT P&P1 CLAMP OPEN" : Bool;
      "X14-2 JR OUT P&P1 CLAMP CLOSE" : Bool;
      "X16-1 JR OUT P&P1 CLAMP OPEN/CLOSE PRESSURE SENSOR" : Bool;
      "X16-2 JR OUT P&P1 Z-AXIS SAFETY PIN LOADING SENSOR" : Bool;
   END_VAR
BEGIN
END_DATA_BLOCK

DATA_BLOCK "BK03"   // DB302
// stored: MemoryReserve 100
   VAR
      "X10-1 JR OUT P&P2 Z-AXIS LIMIT SENSOR(-)" : Bool;
      "X10-2 JR OUT P&P2 Z-AXIS HOME SENSOR" : Bool;
      "X12-1 JR OUT P&P2 Z-AXIS LIMT SENSOR(+)" : Bool;
      "X12-2 JR OUT P&P2 STACK DETECT SENSOR" : Bool;
      "X14-1 JR OUT P&P2 CLAMP OPEN" : Bool;
      "X14-2 JR OUT P&P2 CLAMP CLOSE" : Bool;
      "X16-1 OUT P&P GRIPPER 2ND OPEN/CLOSE PRESSURE SENSOR" : Bool;
      "X16-2 OUT P&P GRIPPER 2ND Z-AXIS SAFETY PIN LOADING SENSOR" : Bool;
   END_VAR
BEGIN
END_DATA_BLOCK

DATA_BLOCK "BK04"   // DB40116
// stored: MemoryReserve 100
   VAR
      "X10-1 STACK #1 NG CLAMP MOVER OPEN" : Bool;
      "X11-1 STACK #1 NG CLAMP RIGHT OPEN" : Bool;
      "X12-1 STACK #1 NG CLAMP LEFT OPEN" : Bool;
      "X13-1 STAKC #1 NG CLAMP Z-AXIS UP" : Bool;
      "X14-1 STAKC #1 NG CLAMP MOVER BACKWARD" : Bool;
      "X15-1 STACK #1 NG BOX LIFT DOWN" : Bool;
      "X16-1 STACK #1 NG BOX LOCK DOWN" : Bool;
      "X17-1 STACK 1 NG BOX FULL SENSOR" : Bool;
      "X10-2 STACK #1 NG CLAMP MOVER CLOSE" : Bool;
      "X11-2 STACK #1 NG CLAMP RIGHT CLOSE" : Bool;
      "X12-2 STACK #1 NG CLAMP LEFT CLOSE" : Bool;
      "X13-2 STAKC #1 NG CLAMP Z-AXIS DOWN" : Bool;
      "X14-2 STAKC #1 NG CLAMP MOVER FORWARD" : Bool;
      "X15-2 STACK #1 NG BOX LIFT UP" : Bool;
      "X16-2 STACK #1 NG BOX LOCK UP" : Bool;
      "X17-2 SPARE" : Bool;
   END_VAR
BEGIN
END_DATA_BLOCK

DATA_BLOCK "BK05"   // DB231
// stored: MemoryReserve 100
   VAR
      "X10-1 STACK #2 NG CLAMP MOVER OPEN" : Bool;
      "X11-1 STACK #2 NG CLAMP LEFT OPEN" : Bool;
      "X12-1 STACK #2 NG CLAMP RIGHT OPEN" : Bool;
      "X13-1 STAKC #2 NG CLAMP Z-AXIS UP" : Bool;
      "X14-1 STAKC #2 NG CLAMP MOVER BACKWARD" : Bool;
      "X15-1 STACK #2 NG BOX LIFT DOWN" : Bool;
      "X16-1 STACK #2 NG BOX LOCK DOWN" : Bool;
      "X17-1 STACK # NG BOX FULL SENSOR" : Bool;
      "X10-2 STACK #2 NG BOX LIFT DOWN" : Bool;
      "X11-2 STACK #2 NG CLAMP LEFT CLOSE" : Bool;
      "X12-2 STACK #2 NG CLAMP RIGHT CLOSE" : Bool;
      "X13-2 STAKC #2 NG CLAMP Z-AXIS DOWN" : Bool;
      "X14-2 STAKC #2 NG CLAMP MOVER FORWARD" : Bool;
      "X15-2 STACK #2 NG BOX LIFT UP" : Bool;
      "X16-2 STACK #2 NG BOX LOCK UP" : Bool;
      "X17-2 SPARE" : Bool;
   END_VAR
BEGIN
END_DATA_BLOCK

DATA_BLOCK "BK06"   // DB232
// stored: MemoryReserve 100
   VAR
      "X10-1 TOP TAPE DIAMETER SENSOR" : Bool;
      "X11-1 TOP TAPE CUTTER UP" : Bool;
      "X12-1 TOP TAPE CUTTER CLAMP UP" : Bool;
      "X13-1 TOP TAPE CLAMP OPEN" : Bool;
      "X14-1 TOP TAPE TENSION BACKWARD" : Bool;
      "X15-1 TOP TAPE LOADING BACKWARD" : Bool;
      "X16-1 SPARE" : Bool;
      "X17-1 SPARE" : Bool;
      "X10-2 SPARE" : Bool;
      "X11-2 TOP TAPE CUTTER DOWN" : Bool;
      "X12-2 TOP TAPE CUTTER CLAMP DOWN" : Bool;
      "X13-2 TOP TAPE CLAMP CLOSE" : Bool;
      "X14-2 TOP TAPE TENSION FORWARD" : Bool;
      "X15-2 TOP TAPE LOADING FORWARD" : Bool;
      "X16-2 SPARE" : Bool;
      "X17-2 SPARE" : Bool;
   END_VAR
BEGIN
END_DATA_BLOCK

DATA_BLOCK "BK07"   // DB233
// stored: MemoryReserve 100
   VAR
      "X10-1 TAPE ATTACHMENT VACUUM PRESSURE SWITCH" : Bool;
      "X10-2 SPARE" : Bool;
      "X12-1 TOP TAPE ATTACHMENT UP" : Bool;
      "X12-2 TOP TAPE ATTACHMENT DOWN" : Bool;
      "X14-1 TOP TAPING X-AXIS LIMIT SENSOR(-)" : Bool;
      "X14-2 TOP TAPING X-AXIS HOMING SENSOR" : Bool;
      "X16-1 TOP TAPING X-AXIS LIMIT SENSOR(+)" : Bool;
      "X16-2 SPARE" : Bool;
   END_VAR
BEGIN
END_DATA_BLOCK

DATA_BLOCK "BK08"   // DB234
// stored: MemoryReserve 100
   VAR
      "X10-1 TOP TAPE CLAMP TOP LEFT UP" : Bool;
      "X11-1 TOP TAPE CLAMP TOP CENTER UP" : Bool;
      "X12-1 TOP TAPE CLAMP TOP RIGHT UP" : Bool;
      "X13-1 TOP TAPE ATTACHMENT VACUUM PRESSURE SWITCH" : Bool;
      "X14-1 TOP TAPE CLAMP BTM DOWN" : Bool;
      "X15-1 TOP TAPING Y-AXIS LIMIT SENSOR(-)" : Bool;
      "X16-1 TOP TAPING Y-AXIS LIMIT SENSOR(+)" : Bool;
      "X17-1 TOP TAPE FIX STAGE STACK DETECT SENSOR" : Bool;
      "X10-2 TOP TAPE CLAMP TOP LEFT DOWN" : Bool;
      "X11-2 TOP TAPE CLAMP TOP CENTER DOWN" : Bool;
      "X12-2 TOP TAPE CLAMP TOP RIGHT DOWN" : Bool;
      "X13-2 SPARE" : Bool;
      "X14-2 TOP TAPE CLAMP BTM UP" : Bool;
      "X15-2 TOP TAPING Y-AXIS HOME SENSOR" : Bool;
      "X16-2 SPARE" : Bool;
      "X17-2 SPARE" : Bool;
   END_VAR
BEGIN
END_DATA_BLOCK

DATA_BLOCK "BK09"   // DB235
// stored: MemoryReserve 100
   VAR
      "X10-1 SIDE TAPE CUTTER BACKWARD" : Bool;
      "X11-1 SIDE TAPE CUTTER CLAMP BACKWARD" : Bool;
      "X12-1 SIDE TAPE CLAMP OPEN" : Bool;
      "X13-1 SIDE TAPE TENSION BACKWARD" : Bool;
      "X14-1 SIDE TAPE LOADING BACKWARD" : Bool;
      "X15-1 SIDE TAPE DIAMETER SENSOR" : Bool;
      "X16-1 SPARE" : Bool;
      "X17-1 SPARE" : Bool;
      "X10-2 SIDE TAPE CUTTER FORWARD" : Bool;
      "X11-2 SIDE TAPE CUTTER CLAMP FORWARD" : Bool;
      "X12-2 SIDE TAPE CLAMP CLOSE" : Bool;
      "X13-2 SIDE TAPE TENSION FORWARD" : Bool;
      "X14-2 SIDE TAPE LOADING FORWARD" : Bool;
      "X15-2 SPARE" : Bool;
      "X16-2 SPARE" : Bool;
      "X17-2 SPARE" : Bool;
   END_VAR
BEGIN
END_DATA_BLOCK

DATA_BLOCK "BK10"   // DB236
// stored: MemoryReserve 100
   VAR
      "X10-1 SIDE TAPE Attachment LEFT BACKWARD" : Bool;
      "X11-1 SIDE TAPE Attachment RIGHT BACKWARD" : Bool;
      "X12-1 SIDE TAPE Attachment 1 TOP VACCUM PRESSURE SWITCH" : Bool;
      "X13-1 SIDE TAPE Attachment 2 TOP VACCUM PRESSURE SWITCH" : Bool;
      "X14-1 SIDE TAPE ATTACHEMNT LEFT PRESSURE SWITCH" : Bool;
      "X15-1 SIDE TAPE Attachment BTM BACKWARD" : Bool;
      "X16-1 SIDE TAPING Y-AYIS LIMIT SENSOR(-)" : Bool;
      "X17-1 SIDE TAPING Y-AYIS LIMIT SENSOR(+)" : Bool;
      "X10-2 SIDE TAPE Attachment LEFT FORWARD" : Bool;
      "X11-2 SIDE TAPE Attachment RIGHT FORWARD" : Bool;
      "X12-2 SIDE TAPE Attachment 1 BTM VACCUM PRESSURE SWITCH" : Bool;
      "X13-2 SIDE TAPE Attachment 2 BTM VACCUM PRESSURE SWITCH" : Bool;
      "X14-2 SIDE TAPE ATTACHMENT RIGHT PRESSURE SWITCH" : Bool;
      "X15-2 SIDE TAPE Attachment BTM FORWARD" : Bool;
      "X16-2 SIDE TAPING Y-AYIS HOME SENSOR" : Bool;
      "X17-2 SPARE" : Bool;
   END_VAR
BEGIN
END_DATA_BLOCK

DATA_BLOCK "BK11"   // DB237
// stored: MemoryReserve 100
   VAR
      "X10-1 SIDE TAPING X-AXIS LIMIT SENSOR(-)" : Bool;
      "X11-1 SIDE TAPING X-AXIS LIMIT SENSOR(+)" : Bool;
      "X12-1 JR FIX STAGE X-AXIS LIMIT SENSOR(-)" : Bool;
      "X13-1 JR FIX STAGE X-AXIS LIMIT SENSOR(+)" : Bool;
      "X14-1 JR FIX STAGE C-AXIS LIMIT SENSOR(-)" : Bool;
      "X15-1 JR FIX STAGE C-AXIS LIMIT SENSOR(+)" : Bool;
      "X16-1 STACK DETECT SENSOR" : Bool;
      "X17-1 SIDE TAPE FIX STAGE OPEN" : Bool;
      "X10-2 SIDE TAPING X-AXIS HOME SENSOR" : Bool;
      "X11-2 SPARE" : Bool;
      "X12-2 JR FIX STAGE X-AXIS HOMING SENSOR" : Bool;
      "X13-2 SPARE" : Bool;
      "X14-2 JR FIX STAGE X-AXIS HOMING SENSOR" : Bool;
      "X15-2 SPARE" : Bool;
      "X16-2 SIDE TAPE CLAMP SAFETY PIN LOADING SENSOR" : Bool;
      "X17-2 SIDE TAPE FIX STAGE CLOSE" : Bool;
   END_VAR
BEGIN
END_DATA_BLOCK

DATA_BLOCK "BK12"   // DB238
// stored: MemoryReserve 100
   VAR
      "X10-1 SPARE" : Bool;
      "X11-1 SPARE" : Bool;
      "X12-1 HP STAGE LIFT #1 FRONT DOWN" : Bool;
      "X13-1 HP STAGE LIFT #1 REAR DOWN" : Bool;
      "X14-1 HP STACK DETECT SENSOR 1" : Bool;
      "X15-1 HP STAGE 1 SAFETY PIN LOADING SENSOR" : Bool;
      "X16-1 SPARE" : Bool;
      "X17-1 SPARE" : Bool;
      "X10-2 SPARE" : Bool;
      "X11-2 SPARE" : Bool;
      "X12-2 HP STAGE LIFT #1 FRONT UP" : Bool;
      "X13-2 HP STAGE LIFT #1 REAR UP" : Bool;
      "X14-2 SPARE" : Bool;
      "X15-2 SPARE" : Bool;
      "X16-2 SPARE" : Bool;
      "X17-2 SPARE" : Bool;
   END_VAR
BEGIN
END_DATA_BLOCK

DATA_BLOCK "BK13"   // DB249
// stored: MemoryReserve 100
   VAR
      "X10-1 SPARE" : Bool;
      "X11-1 SPARE" : Bool;
      "X12-1 HP STAGE LIFT #2 FRONT DOWN" : Bool;
      "X13-1 HP STAGE LIFT #2 REAR DOWN" : Bool;
      "X14-1 HP STACK DETECT SENSOR 2" : Bool;
      "X15-1 HP STAGE 2 SAFETY PIN LOADING SENSOR" : Bool;
      "X16-1 SPARE" : Bool;
      "X17-1 THICKNESS TEST SENSOR AMP POWER" : Bool;
      "X10-2 SPARE" : Bool;
      "X11-2 SPARE" : Bool;
      "X12-2 HP STAGE LIFT #2 FRONT UP" : Bool;
      "X13-2 HP STAGE LIFT #2 REAR UP" : Bool;
      "X14-2 SPARE" : Bool;
      "X15-2 SPARE" : Bool;
      "X16-2 SPARE" : Bool;
      "X17-2 SPARE" : Bool;
   END_VAR
BEGIN
END_DATA_BLOCK

DATA_BLOCK "BK14"   // DB258
// stored: MemoryReserve 100
   VAR
      "X10-1 HIPOT TAB CONTACTOR BACKWARD" : Bool;
      "X11-1 HIPOT TAB CONTACTOR LEFT OPEN" : Bool;
      "X12-1 HIPOT TAB CONTACTOR RIGHT OPEN" : Bool;
      "X13-1 SPARE" : Bool;
      "X14-1 SPARE" : Bool;
      "X15-1 HIPOT&THICKNESS STAGE LIFT FRONT DOWN" : Bool;
      "X16-1 HIPOT&THICKNESS STAGE LIFT REAR DOWN" : Bool;
      "X17-1 SPARE" : Bool;
      "X10-2 HIPOT TAB CONTACTOR FORWARD" : Bool;
      "X11-2 HIPOT TAB CONTACTOR LEFT CLOSE" : Bool;
      "X12-2 HIPOT TAB CONTACTOR RIGHT CLOSE" : Bool;
      "X13-2 SPARE" : Bool;
      "X14-2 SPARE" : Bool;
      "X15-2 INSPECTION STAGE LIFT FRONT UP" : Bool;
      "X16-2 INSPECTION STAGE LIFT REAR UP" : Bool;
      "X17-2 SPARE" : Bool;
   END_VAR
BEGIN
END_DATA_BLOCK

DATA_BLOCK "BK15"   // DB259
// stored: MemoryReserve 100
   VAR
      "X10-1 HIPOT&THICKNESS Z-AXIS LIMIT SENSOR(-)" : Bool;
      "X11-1 HIPOT&THICKNESS Z-AXIS LIMIT SENSOR(+)" : Bool;
      "X12-1 HIPOT&THICKNESS STACK DETECT SENSOR" : Bool;
      "X13-1 HI-POT SAFETY PIN LOADING SENSOR" : Bool;
      "X14-1 SPARE" : Bool;
      "X15-1 SPARE" : Bool;
      "X16-1 SPARE" : Bool;
      "X17-1 SPARE" : Bool;
      "X10-2 HIPOT&THICKNESS Z-AXIS HOME SENSOR" : Bool;
      "X11-2 SPARE" : Bool;
      "X12-2 SPARE" : Bool;
      "X13-2 SPARE" : Bool;
      "X14-2 SPARE" : Bool;
      "X15-2 SPARE" : Bool;
      "X16-2 SPARE" : Bool;
      "X17-2 SPARE" : Bool;
   END_VAR
BEGIN
END_DATA_BLOCK

DATA_BLOCK "BK16"   // DB260
// stored: MemoryReserve 100
   VAR
      "X10-1 FINAL VISION STAGE LIFT UP" : Bool;
      "X10-2 FINAL VISION STAGE LIFT DOWN" : Bool;
      "X12-1 FINAL VISION LIGHT UP" : Bool;
      "X12-2 FINAL VISION LIGHT DOWN" : Bool;
      "X14-1 FINAL VISION STAGE DETECT SENSOR" : Bool;
      "X14-2 SPARE" : Bool;
      "X16-1 SPARE" : Bool;
      "X16-2 SPARE" : Bool;
   END_VAR
BEGIN
END_DATA_BLOCK

DATA_BLOCK "BK17"   // DB263
// stored: MemoryReserve 100
   VAR
      "X10-1 LASER MARKING COVER UP" : Bool;
      "X10-2 LASER MARKING COVER DOWN" : Bool;
      "X12-1 LASER MARKING Stage Lift UP" : Bool;
      "X12-2 LASER MARKING Stage Lift DOWN" : Bool;
      "X14-1 SPARE" : Bool;
      "X14-2 LASER MARKING STACK DETECT SENSOR" : Bool;
      "X16-1 SPARE" : Bool;
      "X16-2 SPARE" : Bool;
   END_VAR
BEGIN
END_DATA_BLOCK

DATA_BLOCK "BK18"   // DB264
// stored: MemoryReserve 100
   VAR
      "X10-1 WEIGHT NG CLAMP MOVER OPEN" : Bool;
      "X11-1 WEIGHT NG CLAMP LEFT OPEN" : Bool;
      "X12-1 WEIGHT NG CLAMP RIGHT OPEN" : Bool;
      "X13-1 WEIGHT NG CLAMP Z-AXIS UP" : Bool;
      "X14-1 WEIGHT NG CLAMP MOVER BACKWARD" : Bool;
      "X15-1 WEIGHT NG BOX LIFT DOWN" : Bool;
      "X16-1 WEIGHT NG BOX LOCK DOWN" : Bool;
      "X17-1 STACK NG FULL SENSOR" : Bool;
      "X10-2 WEIGHT NG CLAMP MOVER CLOSE" : Bool;
      "X11-2 WEIGHT NG CLAMP LEFT CLOSE" : Bool;
      "X12-2 WEIGHT NG CLAMP RIGHT CLOSE" : Bool;
      "X13-2 WEIGHT NG CLAMP Z-AXIS DOWN" : Bool;
      "X14-2 WEIGHT NG CLAMP MOVER FORWARD" : Bool;
      "X15-2 WEIGHT NG BOX LIFT UP" : Bool;
      "X16-2 WEIGHT NG BOX LOCK UP" : Bool;
      "X17-2 SPARE" : Bool;
   END_VAR
BEGIN
END_DATA_BLOCK

DATA_BLOCK "BK19"   // DB266
// stored: MemoryReserve 100
   VAR
      "X10-1 SPARE" : Bool;
      "X10-2 SPARE" : Bool;
      "X12-1 SPARE" : Bool;
      "X12-2 SPARE" : Bool;
      "X14-1 WEIGHT DETECT SENSOR" : Bool;
      "X14-2 SPARE" : Bool;
      "X16-1 MAIN VALVE DIGITAL PRESSURE SWITCH OUT1" : Bool;
      "X16-2 MAIN VALVE DIGITAL PRESSURE SWITCH OUT2" : Bool;
   END_VAR
BEGIN
END_DATA_BLOCK

DATA_BLOCK "BK20"   // DB267
// stored: MemoryReserve 100
   VAR
      "X10-1 INS TRANSFER P&P1 X-AXIS LIMIT SENSOR(-)" : Bool;
      "X11-1 INS TRANSFER P&P1 X-AXIS LIMIT SENSOR(+)" : Bool;
      "X12-1 INS TRANSFER P&P2 X-AXIS LIMIT SENSOR(-)" : Bool;
      "X13-1 INS TRANSFER P&P2 X-AXIS LIMIT SENSOR(+)" : Bool;
      "X14-1 SPARE" : Bool;
      "X15-1 SPARE" : Bool;
      "X16-1 SPARE" : Bool;
      "X17-1 SPARE" : Bool;
      "X10-2 INS TRANSFER P&P1 X-AXIS HOMING SENSOR" : Bool;
      "X11-2 SPARE" : Bool;
      "X12-2 INS TRANSFER P&P2 X-AXIS HOMING SENSOR" : Bool;
      "X13-2 SPARE" : Bool;
      "X14-2 SPARE" : Bool;
      "X15-2 SPARE" : Bool;
      "X16-2 SPARE" : Bool;
      "X17-2 SPARE" : Bool;
   END_VAR
BEGIN
END_DATA_BLOCK

DATA_BLOCK "BK21"   // DB268
// stored: MemoryReserve 100
   VAR
      "X10-1 INS TRANSFER P&P1 Y-AXIS LIMIT SENSOR(-)" : Bool;
      "X11-1 INS TRANSFER P&P1 Y-AXIS LIMIT SENSOR(+)" : Bool;
      "X12-1 INS TRANSFER P&P1 Z-AXIS LIMIT SENSOR(-)" : Bool;
      "X13-1 INS TRANSFER P&P1 Z-AXIS LIMIT SENSOR(+)" : Bool;
      "X14-1 INS TRANSFER P&P1 CLAMP OPEN SENSOR" : Bool;
      "X15-1 INS TRANSFER P&P1 CLAMP STACK DETECT SENSOR" : Bool;
      "X16-1 INS TRANSFER P&P1 Z-AXIS SAFETY PIN LOADING SENSOR" : Bool;
      "X17-1 STACK NG BOX DETECT SENSOR" : Bool;
      "X10-2 INS TRANSFER P&P1 Y-AXIS HOMING SENSOR" : Bool;
      "X11-2 SPARE" : Bool;
      "X12-2 INS TRANSFER P&P1 Z-AXIS HOMING SENSOR" : Bool;
      "X13-2 SPARE" : Bool;
      "X14-2 INS TRANSFER P&P1 CLAMP CLOSE SENSOR" : Bool;
      "X15-2 INS TRANSFER P&P1 CLAMP OPEN/CLOSE PRESSURE SENSOR" : Bool;
      "X16-2 SPARE" : Bool;
      "X17-2 SPARE" : Bool;
   END_VAR
BEGIN
END_DATA_BLOCK

DATA_BLOCK "BK22"   // DB269
// stored: MemoryReserve 100
   VAR
      "X10-1 INS TRANSFER P&P2 Y-AXIS LIMIT SENSOR(-)" : Bool;
      "X11-1 INS TRANSFER P&P2 Y-AXIS LIMIT SENSOR(+)" : Bool;
      "X12-1 INS TRANSFER P&P2 Z-AXIS LIMIT SENSOR(-)" : Bool;
      "X13-1 INS TRANSFER P&P2 Z-AXIS LIMIT SENSOR(+)" : Bool;
      "X14-1 INS TRANSFER P&P2 CLAMP OPEN SENSOR" : Bool;
      "X15-1 INS TRANSFER P&P2 CLAMP STACK DETECT SENSOR" : Bool;
      "X16-1 INS TRANSFER P&P2 Z-AXIS SAFETY PIN LOADING SENSOR" : Bool;
      "X17-1 SPARE" : Bool;
      "X10-2 INS TRANSFER P&P2 Y-AXIS HOMING SENSOR" : Bool;
      "X11-2 SPARE" : Bool;
      "X12-2 PROCESS P&P Z-AXIS HEAD2 HOMING SENSOR" : Bool;
      "X13-2 SPARE" : Bool;
      "X14-2 INS TRANSFER P&P2 CLAMP CLOSE SENSOR" : Bool;
      "X15-2 INS TRANSFER P&P2 CLAMP OPEN/CLOSE PRESSURE SENSOR" : Bool;
      "X16-2 SPARE" : Bool;
      "X17-2 SPARE" : Bool;
   END_VAR
BEGIN
END_DATA_BLOCK

DATA_BLOCK "BK23"   // DB270
// stored: MemoryReserve 100
   VAR
      "X10-1 JR Unloading P&P Y-AXIS LIMIT SENSOR(-)" : Bool;
      "X11-1 JR Unloading P&P Y-AXIS LIMIT SENSOR(+)" : Bool;
      "X12-1 JR Unloading P&P Z-AXIS LIMIT SENSOR(-)" : Bool;
      "X13-1 JR Unloading P&P Z-AXIS LIMIT SENSOR(+)" : Bool;
      "X14-1 JR Unloading P&P C-AXIS LIMIT SENSOR(-)" : Bool;
      "X15-1 JR Unloading P&P C-AXIS LIMIT SENSOR(+)" : Bool;
      "X16-1 JR Unloading P&P CLAMP OPEN SENSOR" : Bool;
      "X17-1 JR Unloading P&P CLAMP STACK DETECT SENSOR" : Bool;
      "X10-2 JR Unloading P&P Y-AXIS HOMING SENSOR" : Bool;
      "X11-2 SPARE" : Bool;
      "X12-2 JR Unloading P&P Z-AXIS HOMING SENSOR" : Bool;
      "X13-2 SPARE" : Bool;
      "X14-2 JR Unloading P&P C-AXIS HOMING SENSOR" : Bool;
      "X15-2 SPARE" : Bool;
      "X16-2 JR Unloading P&P CLAMP CLOSE SENSOR" : Bool;
      "X17-2 JR Unloading P&P Z-AXIS SAFETY PIN LOADING SENSOR" : Bool;
   END_VAR
BEGIN
END_DATA_BLOCK

DATA_BLOCK "BK24"   // DB271
// stored: MemoryReserve 100
   VAR
      "X10-1 SIDE TAPE ATTACHMENT #1 TOP VACUUM ON" : Bool;
      "X10-2 SIDE TAPE ATTACHMENT #1 TOP VACUUM OFF" : Bool;
      "X12-1 SIDE TAPE ATTACHMENT #1 BTM VACUUM ON" : Bool;
      "X12-2 SIDE TAPE ATTACHMENT #1 BTM VACUUM OFF" : Bool;
      "X14-1 SIDE TAPE ATTACHMENT #2 TOP VACUUM ON" : Bool;
      "X14-2 SIDE TAPE ATTACHMENT #2 TOP VACUUM OFF" : Bool;
      "X16-1 SIDE TAPE ATTACHMENT #2 BTM VACUUM ON" : Bool;
      "X16-2 SIDE TAPE ATTACHMENT #2 BTM VACUUM OFF" : Bool;
   END_VAR
BEGIN
END_DATA_BLOCK

DATA_BLOCK "BK25"   // DB272
// stored: MemoryReserve 100
   VAR
      "X10-1 TOP TAPE ATTACHMENT #1 VACUUM ON" : Bool;
      "X10-2 TOP TAPE ATTACHMENT #1 VACUUM OFF" : Bool;
      "X12-1 SPARE" : Bool;
      "X12-2 SPARE" : Bool;
      "X14-1 SPARE" : Bool;
      "X14-2 SPARE" : Bool;
      "X16-1 SPARE" : Bool;
      "X16-2 SPARE" : Bool;
   END_VAR
BEGIN
END_DATA_BLOCK

DATA_BLOCK "MP101"   // DB181
// stored: MemoryReserve 100
   VAR
      "KISTLER 100KN PRESS POWER TRIPPED E202CB" : Bool;
      "KISTLER 100KN PRESS POWER TRIPPED E208CB" : Bool;
      "KISTLER 30KN PRESS POWER TRIPPED E214CB" : Bool;
      SPARE : Bool;
      SPARE_1 : Bool;
      "E8404PWS CONTROLLER POWER SMPS AC POWER TRIPPED E320CB" : Bool;
      "E8704PWS SAFETY POWER SMPS AC POWER TRIPPED E326CB" : Bool;
      "E8804PWS CONTRL POWER SMPS AC POWER TRIPPED E332CB" : Bool;
      "PROCESSOR POWER ON TIPPRED E4120CB" : Bool;
      "PROGRAMING POWER OUTLET TRPPED E4126CB" : Bool;
      SPARE_2 : Bool;
      "PANEL LED POWER TRIPPED E4304CB" : Bool;
      SPARE_3 : Bool;
      "PLC POWER SMPS DC OK E4404PWS" : Bool;
      "CONTROL LEVEL HUB POWER TRIPPED E4420CB" : Bool;
      "MAIN HMI POWER TRIPPED E4426CB" : Bool;
      "PORTABLE HMI POWER TIPPED E4432CB" : Bool;
      "PORTABLE HMI POWER TIPPED E4456CB" : Bool;
      "120VAC HEATER-1 POWER TR PRIMARY TRIPPED E5100CB" : Bool;
      SPARE_4 : Bool;
      SPARE_5 : Bool;
      "UPPER 1-1 HEATER POWER TRIPPED E5156CB" : Bool;
      "UPPER 1-2 HEATER POWER TRIPPED E5162CB" : Bool;
      "LOWER 1-1 HEATER POWER TRIPPED E5168CB" : Bool;
      "LOWER 1-2 HEATER POWER TRIPPED E5174CB" : Bool;
      "LOWER 1-3 HEATER POWER TRIPPED E5180CB" : Bool;
      SPARE_6 : Bool;
      "120VAC HEATER-2 POWER TR PRIMARY TRIPPED E6100CB" : Bool;
      SPARE_7 : Bool;
      SPARE_8 : Bool;
      "UPPER 2-1 HEATER POWER TRIPPED E6156CB" : Bool;
      "UPPER 2-2 HEATER POWER TRIPPED E6162CB" : Bool;
   END_VAR
BEGIN
END_DATA_BLOCK

DATA_BLOCK "MP102"   // DB304
// stored: MemoryReserve 100
   VAR
      "LOWER 2-1 HEATER POWER TRIPPED E6168CB" : Bool;
      "LOWER 2-2 HEATER POWER TRIPPED E6174CB" : Bool;
      "LOWER 2-3 HEATER POWER TRIPPED E6180CB" : Bool;
      "VISION LIGHT CONTROLLER POWER STRIP OUTLET POWER TRIPPED E7184CB" : Bool;
      "120VAC CONTROL POWER TR PRIMARY TRIPPED E7100CB" : Bool;
      "120VAC CONTROL POWER TR SECONDARY TRIPPED E7110CB" : Bool;
      "CONTROL POWER ON TRIPPED E7116CB" : Bool;
      "MOTOR PANEL CONTROL POWER TRIPPED E7154CB" : Bool;
      "WEIGHT TESTER POWER STRIP OUTLET POWER TRIPPED E7160CB" : Bool;
      "VISION MONITOR & MCU POWER STRIP OUTLET POWER TRIPPED E7166CB" : Bool;
      "QR LASER MARKING TRIPPED E7172CB" : Bool;
      "HI-POT TESTER POWER STRIP OUTLET POWER TRIPPED E7178CB" : Bool;
      "FFU-1 POWER TRIPPED E7222CB" : Bool;
      "UPPER 1-1 TEMPERATURE CONTROLLER POWER TRIPPED E5206CB" : Bool;
      "UPPER 1-2 TEMPERATURE CONTROLLER POWER TRIPPED E5212CB" : Bool;
      "LOWER 1-1 TEMPERATURE CONTROLLER POWER TRIPPED E5218CB" : Bool;
      "LOWER 1-2 TEMPERATURE CONTROLLER POWER TRIPPED E5224CB" : Bool;
      "LOWER 1-3 TEMPERATURE CONTROLLER POWER TRIPPED E5230CB" : Bool;
      "UPPER 2-1 TEMPERATURE CONTROLLER POWER TRIPPED E6206CB" : Bool;
      "UPPER 2-2 TEMPERATURE CONTROLLER POWER TRIPPED E6212CB" : Bool;
      "LOWER 2-1 TEMPERATURE CONTROLLER POWER TRIPPED E6218CB" : Bool;
      "LOWER 2-2 TEMPERATURE CONTROLLER POWER TRIPPED E6224CB" : Bool;
      "LOWER 2-3 TEMPERATURE CONTROLLER POWER TRIPPED E6230CB" : Bool;
      SPARE : Bool;
      "CONTROL POWER SMPS DC OK E8104PWS" : Bool;
      "ET200MP I/O OUTPUT POWER TRIPPED E8154CB" : Bool;
      "JUNCTION BOX CONTROL POWER TRIPPED E8180CB" : Bool;
      "CLASS 2 SMPS POWER TRIPPED E8204CB" : Bool;
      "CLASS 2 SMPS MONITORING E8206PWS" : Bool;
      "ET200ECO PN-1 POWER TRIPPED E8220CB" : Bool;
      "ET200ECO PN-2 POWER TRIPPED E8224CB" : Bool;
      "ET200ECO PN-3 POWER TRIPPED E8228CB" : Bool;
   END_VAR
BEGIN
END_DATA_BLOCK

DATA_BLOCK "MP103"   // DB305
// stored: MemoryReserve 100
   VAR
      "ET200ECO PN-4 POWER TRIPPED E8232CB" : Bool;
      "PANEL FAN POWER TRIPPED E8304CB" : Bool;
      SPARE : Bool;
      "CONTROLLER POWER SMPS DC OK E8404PWS" : Bool;
      "CONTROLLER DC POWER TRIPPED E8406CB" : Bool;
      "KISTLER CONTROL POWER TRIPPED E8416CB" : Bool;
      "MANIFOLD-1 POWER TRIPPED E8422CB" : Bool;
      "MANIFOLD-2 POWER TRIPPED E8430CB" : Bool;
      "QR READER POWER TRIPPED E8456CB" : Bool;
      "QR READER POWER TRIPPED E8462CB" : Bool;
      "HANDY QR READER POWER TRIPPED E8468CB" : Bool;
      "PROFINET CONVERTER POWER TRIPPED E8474CB" : Bool;
      "MONITORING RELAY POWER TRIPPED E8504CB" : Bool;
      SPARE_1 : Bool;
      "SAFETY POWER SMPS DC OK E8704PWS" : Bool;
      "SAFETY DC POWER TRIPPED E8706CB" : Bool;
      "ET200SP I/O SAFETY POWER TRIPPED E8716CB" : Bool;
      "JUNCTION BOX CONTROL POWER TRIPPED E8736CB" : Bool;
      "ET200ECO PN SAFETYT-1 POWER TRIPPED E8756CB" : Bool;
      "ET200ECO PN SAFETYT-2 POWER TRIPPED E8762CB" : Bool;
      SPARE_2 : Bool;
      "CONTROL POWER SMPS DC OK E8804PWS" : Bool;
      "CONTROL DC POWER TRIPPED E8806CB" : Bool;
      "JUNCTION BOX CONTROL POWER TRIPPED E8816CB" : Bool;
      "DRIVE-CLIQ HUB POWER TRIPPED E8822CB" : Bool;
      "EQUIPMENT LED POWER TRIPPED E8828CB" : Bool;
      SPARE_3 : Bool;
      SPARE_4 : Bool;
      SPARE_5 : Bool;
      SPARE_6 : Bool;
      SPARE_7 : Bool;
      SPARE_8 : Bool;
   END_VAR
BEGIN
END_DATA_BLOCK

DATA_BLOCK "MP104"   // DB307
// stored: MemoryReserve 100
   VAR
      "UPPER 1-1 HEATER MONITOR SIGNAL ON" : Bool;
      "UPPER 1-2 HEATER MONITOR SIGNAL ON" : Bool;
      "LOWER 1-1 HEATER MONITOR SIGNAL ON" : Bool;
      "LOWER 1-2 HEATER MONITOR SIGNAL ON" : Bool;
      "LOWER 1-3 HEATER MONITOR SIGNAL ON" : Bool;
      "UPPER 2-1 HEATER MONITOR SIGNAL ON" : Bool;
      "UPPER 2-2 HEATER MONITOR SIGNAL ON" : Bool;
      "LOWER 2-1 HEATER MONITOR SIGNAL ON" : Bool;
      "LOWER 2-2 HEATER MONITOR SIGNAL ON" : Bool;
      "LOWER 2-3 HEATER MONITOR SIGNAL ON" : Bool;
      SPARE : Bool;
      SPARE_1 : Bool;
      SPARE_2 : Bool;
      SPARE_3 : Bool;
      SPARE_4 : Bool;
      SPARE_5 : Bool;
      SPARE_6 : Bool;
      SPARE_7 : Bool;
      SPARE_8 : Bool;
      SPARE_9 : Bool;
      SPARE_10 : Bool;
      SPARE_11 : Bool;
      SPARE_12 : Bool;
      SPARE_13 : Bool;
      SPARE_14 : Bool;
      SPARE_15 : Bool;
      SPARE_16 : Bool;
      SPARE_17 : Bool;
      SPARE_18 : Bool;
      SPARE_19 : Bool;
      SPARE_20 : Bool;
      SPARE_21 : Bool;
   END_VAR
BEGIN
END_DATA_BLOCK

DATA_BLOCK "MP105"   // DB306
// stored: MemoryReserve 100
   VAR
      "EQUIPMENT LED LAMP RELAY ON" : Bool;
      SPARE : Bool;
      SPARE_1 : Bool;
      "CLASS2 SMPS ALARM RESET" : Bool;
      SPARE_2 : Bool;
      SPARE_3 : Bool;
      SPARE_4 : Bool;
      SPARE_5 : Bool;
      "QR MARKER TOWER LAMP 1 ON (RED)" : Bool;
      "QR MARKER TOWER LAMP 2 ON (AMBER)" : Bool;
      "QR MARKER TOWER LAMP 3 ON (GREEN)" : Bool;
      "QR MARKER TOWER LAMP 4 ON (WHITE)" : Bool;
      "QR MARKER TOWER LAMP 5 ON (BLUE)" : Bool;
      "QR MARKER TOWER LAMP BUZZER ON" : Bool;
      SPARE_6 : Bool;
      SPARE_7 : Bool;
      SPARE_8 : Bool;
      SPARE_9 : Bool;
      SPARE_10 : Bool;
      SPARE_11 : Bool;
      SPARE_12 : Bool;
      SPARE_13 : Bool;
      SPARE_14 : Bool;
      SPARE_15 : Bool;
      SPARE_16 : Bool;
      SPARE_17 : Bool;
      SPARE_18 : Bool;
      SPARE_19 : Bool;
      SPARE_20 : Bool;
      SPARE_21 : Bool;
      SPARE_22 : Bool;
      SPARE_23 : Bool;
   END_VAR
BEGIN
END_DATA_BLOCK

DATA_BLOCK "MP106"   // DB308
// stored: MemoryReserve 100
   VAR
      "MANIFOLD-1 SOL POWER MC FEEDBACK" : Bool;
      "MANIFOLD-2 SOL POWER MC FEEDBACK" : Bool;
      "QR LASER MARKING POWER 1 FEEDBACK" : Bool;
      "QR LASER MARKING POWER 2 FEEDBACK" : Bool;
      "FFU POWER MC 1 FEEDBACK" : Bool;
      "FFU POWER MC 2 FEEDBACK" : Bool;
      SPARE : Bool;
      SPARE_1 : Bool;
      SPARE_2 : Bool;
      SPARE_3 : Bool;
      SPARE_4 : Bool;
      SPARE_5 : Bool;
      SPARE_6 : Bool;
      SPARE_7 : Bool;
      SPARE_8 : Bool;
      SPARE_9 : Bool;
      SPARE_20 : Bool;
      SPARE_21 : Bool;
      SPARE_22 : Bool;
      SPARE_23 : Bool;
      SPARE_24 : Bool;
      SPARE_25 : Bool;
      SPARE_10 : Bool;
      SPARE_11 : Bool;
      SPARE_12 : Bool;
      SPARE_13 : Bool;
      SPARE_14 : Bool;
      SPARE_15 : Bool;
      SPARE_16 : Bool;
      SPARE_17 : Bool;
      SPARE_18 : Bool;
      SPARE_19 : Bool;
   END_VAR
BEGIN
END_DATA_BLOCK

DATA_BLOCK "MP107"   // DB309
// stored: MemoryReserve 100
   VAR
      "MANIFOLD-1 SOL POWER MC ON" : Bool;
      "MANIFOLD-2 SOL POWER MC ON" : Bool;
      "QR LASER MARKING POWER ON 1" : Bool;
      "QR LASER MARKING POWER ON 2" : Bool;
      "FFU POWER MC ON 1" : Bool;
      "FFU POWER MC ON 2" : Bool;
      SPARE : Bool;
      SPARE_1 : Bool;
   END_VAR
BEGIN
END_DATA_BLOCK

DATA_BLOCK "MP108"   // DB310
// stored: MemoryReserve 100
   VAR
      "10 TON SERVO PRESS-1 Z-AXIS EMS&STO SIGNAL" : Bool;
      "10 TON SERVO PRESS-1 Z-AXIS - PROBE 1" : Bool;
      "10 TON SERVO PRESS-2 Z-AXIS EMS&STO SIGNAL" : Bool;
      "10 TON SERVO PRESS-2 Z-AXIS - PROBE 1" : Bool;
      "3 TON SERVO PRESS Z-AXIS EMS&STO SIGNAL" : Bool;
      "3 TON SERVO PRESS Z-AXIS - PROBE 1" : Bool;
      SPARE : Bool;
      SPARE_1 : Bool;
   END_VAR
BEGIN
END_DATA_BLOCK

DATA_BLOCK "MP109"   // DB311
// stored: MemoryReserve 100
BEGIN
END_DATA_BLOCK

DATA_BLOCK "PM1"   // DB273
// stored: MemoryReserve 100
   VAR
      "STACK #1 NG CLAMP MOVER CLOSE" : Bool;
      "STACK #1 NG CLAMP MOVER OPEN" : Bool;
      "STACK #1 NG CLAMP RIGHT CLOSE" : Bool;
      "STACK #1 NG CLAMP RIGHT OPEN" : Bool;
      "STACK #1 NG CLAMP LEFT OPEN" : Bool;
      "STACK #1 NG CLAMP LEFT CLOSE" : Bool;
      "STAKC #1 NG CLAMP Z-AXIS UP" : Bool;
      "STAKC #1 NG CLAMP Z-AXIS DOWN" : Bool;
      "STAKC #1 NG CLAMP MOVER FORWARD" : Bool;
      "STAKC #1 NG CLAMP MOVER BACKWARD" : Bool;
      "STACK #1 NG BOX LIFT UP" : Bool;
      "STACK #1 NG BOX LIFT DOWN" : Bool;
      "STACK #1 NG BOX LOCK UP" : Bool;
      "STACK #1 NG BOX LOCK DOWN" : Bool;
      "JR OUT P&P#1 CLAMP CLOSE" : Bool;
      "JR OUT P&P#1 CLAMP OPEN" : Bool;
   END_VAR
BEGIN
END_DATA_BLOCK

DATA_BLOCK "PM10"   // DB284
// stored: MemoryReserve 100
   VAR
      "STACK NG CLAMP MOVER CLOSE" : Bool;
      "STACK NG CLAMP MOVER OPEN" : Bool;
      "STACK NG CLAMP LEFT CLOSE" : Bool;
      "STACK NG CLAMP LEFT OPEN" : Bool;
      "STACK NG CLAMP RIGHT CLOSE" : Bool;
      "STACK NG CLAMP RIGHT OPEN" : Bool;
      "STACK NG CLAMP Z-AXIS UP" : Bool;
      "STACK NG CLAMP Z-AXIS DOWN" : Bool;
      "STACK NG CLAMP MOVER FORWARD" : Bool;
      "STACK NG CLAMP MOVER BACKWARD" : Bool;
      "STACK NG BOX LIFT UP" : Bool;
      "STACK NG BOX LIFT DOWN" : Bool;
      "STACK NG BOX LOCK UP" : Bool;
      "STACK NG BOX LOCK DOWN" : Bool;
      SPARE : Bool;
      SPARE_1 : Bool;
   END_VAR
BEGIN
END_DATA_BLOCK

DATA_BLOCK "PM2"   // DB274
// stored: MemoryReserve 100
   VAR
      "STACK #2 NG CLAMP MOVER CLOSE" : Bool;
      "STACK #2 NG CLAMP MOVER OPEN" : Bool;
      "STACK #2 NG CLAMP LEFT CLOSE" : Bool;
      "STACK #2 NG CLAMP LEFT OPEN" : Bool;
      "STACK #2 NG CLAMP RIGHT CLOSE" : Bool;
      "STACK #2 NG CLAMP RIGHT OPEN" : Bool;
      "STAKC #2 NG CLAMP Z-AXIS UP" : Bool;
      "STAKC #2 NG CLAMP Z-AXIS DOWN" : Bool;
      "STAKC #2 NG CLAMP MOVER FORWARD" : Bool;
      "STAKC #2 NG CLAMP MOVER BACKWARD" : Bool;
      "STACK #2 NG BOX LIFT UP" : Bool;
      "STACK #2 NG BOX LIFT DOWN" : Bool;
      "STACK #2 NG BOX LOCK UP" : Bool;
      "STACK #2 NG BOX LOCK DOWN" : Bool;
      "JR OUT P&P#2 CLAMP CLOSE" : Bool;
      "JR OUT P&P#2 CLAMP OPEN" : Bool;
   END_VAR
BEGIN
END_DATA_BLOCK

DATA_BLOCK "PM3"   // DB277
// stored: MemoryReserve 100
   VAR
      "TOP TAPE CUTTER UP" : Bool;
      "TOP TAPE CUTTER DOWN" : Bool;
      "TOP TAPE CUTTER CLAMP UP" : Bool;
      "TOP TAPE CUTTER CLAMP DOWN" : Bool;
      "TOP TAPE CLAMP OPEN" : Bool;
      "TOP TAPE CLAMP CLOSE" : Bool;
      "TOP TAPE TENSION FORWARD" : Bool;
      "TOP TAPE TENSION BACKWARD" : Bool;
      "TOP TAPE LOADING FORWARD" : Bool;
      "TOP TAPE LOADING BACKWARD" : Bool;
      "TOP TAPE ATTACHMENT UP" : Bool;
      "TOP TAPE ATTACHMENT DOWN" : Bool;
      SPARE : Bool;
      SPARE_1 : Bool;
      SPARE_2 : Bool;
      SPARE_3 : Bool;
   END_VAR
BEGIN
END_DATA_BLOCK

DATA_BLOCK "PM4"   // DB278
// stored: MemoryReserve 100
   VAR
      "TOP TAPE Clamp TOP LEFT UP" : Bool;
      "TOP TAPE Clamp TOP LEFT DOWN" : Bool;
      "TOP TAPE Clamp TOP CENTER UP" : Bool;
      "TOP TAPE Clamp TOP CENTER DOWN" : Bool;
      "TOP TAPE Clamp TOP RIGHT UP" : Bool;
      "TOP TAPE Clamp TOP RIGHT DOWN" : Bool;
      "TOP TAPE Clamp BTM UP" : Bool;
      "TOP TAPE Clamp BTM DOWN" : Bool;
      SPARE : Bool;
      SPARE_1 : Bool;
      SPARE_2 : Bool;
      SPARE_3 : Bool;
      SPARE_4 : Bool;
      SPARE_5 : Bool;
      SPARE_6 : Bool;
      SPARE_7 : Bool;
   END_VAR
BEGIN
END_DATA_BLOCK

DATA_BLOCK "PM5"   // DB279
// stored: MemoryReserve 100
   VAR
      "SIDE TAPE CUTTER FORWARD" : Bool;
      "SIDE TAPE CUTTER BACKWARD" : Bool;
      "SIDE TAPE CUTTER CLAMP FORWARD" : Bool;
      "SIDE TAPE CUTTER CLAMP BACKWARD" : Bool;
      "SIDE TAPE CLAMP CLOSE" : Bool;
      "SIDE TAPE CLAMP OPEN" : Bool;
      "SIDE TAPE TENSION FORWARD" : Bool;
      "SIDE TAPE TENSION BACKWARD" : Bool;
      "SIDE TAPE LOADING FORWARD" : Bool;
      "SIDE TAPE LOADING BACKWARD" : Bool;
      SPARE : Bool;
      SPARE_1 : Bool;
      SPARE_2 : Bool;
      SPARE_3 : Bool;
      SPARE_4 : Bool;
      SPARE_5 : Bool;
   END_VAR
BEGIN
END_DATA_BLOCK

DATA_BLOCK "PM6"   // DB280
// stored: MemoryReserve 100
   VAR
      "SIDE TAPE FIX STAGE CLOSE" : Bool;
      "SIDE TAPE FIX STAGE OPEN" : Bool;
      "SIDE TAPE Attachment LEFT FORWARD" : Bool;
      "SIDE TAPE Attachment LEFT BACKWARD" : Bool;
      "SIDE TAPE Attachment RIGHT FORWARD" : Bool;
      "SIDE TAPE Attachment RIGHT BACKWARD" : Bool;
      "SIDE TAPE Attachment BTM FORWARD" : Bool;
      "SIDE TAPE Attachment BTM BACKWARD" : Bool;
      SPARE : Bool;
      SPARE_1 : Bool;
      SPARE_2 : Bool;
      SPARE_3 : Bool;
      SPARE_4 : Bool;
      SPARE_5 : Bool;
      SPARE_6 : Bool;
      SPARE_7 : Bool;
   END_VAR
BEGIN
END_DATA_BLOCK

DATA_BLOCK "PM7"   // DB281
// stored: MemoryReserve 100
   VAR
      SPARE : Bool;
      SPARE_1 : Bool;
      SPARE_2 : Bool;
      SPARE_3 : Bool;
      SPARE_4 : Bool;
      SPARE_5 : Bool;
      SPARE_6 : Bool;
      SPARE_7 : Bool;
      "HP STAGE LIFT #1 FRONT UP" : Bool;
      "HP STAGE LIFT #1 FRONT DOWN" : Bool;
      "HP STAGE LIFT #1 REAR UP" : Bool;
      "HP STAGE LIFT #1 REAR DOWN" : Bool;
      "HP STAGE LIFT #2 FRONT UP" : Bool;
      "HP STAGE LIFT #2 FRONT DOWN" : Bool;
      "HP STAGE LIFT #2 REAR UP" : Bool;
      "HP STAGE LIFT #2 REAR DOWN" : Bool;
   END_VAR
BEGIN
END_DATA_BLOCK

DATA_BLOCK "PM8"   // DB282
// stored: MemoryReserve 100
   VAR
      "HIPOT TAB CONTACTOR FORWARD" : Bool;
      "HIPOT TAB CONTACTOR BACKWARD" : Bool;
      "HIPOT TAB CONTACTOR LEFT CLOSE" : Bool;
      "HIPOT TAB CONTACTOR LEFT OPEN" : Bool;
      "HIPOT TAB CONTACTOR RIGHT CLOSE" : Bool;
      "HIPOT TAB CONTACTOR RIGHT OPEN" : Bool;
      SPARE : Bool;
      SPARE_1 : Bool;
      SPARE_2 : Bool;
      SPARE_3 : Bool;
      "HIPOT & THICKNESS STAGE LIFT FRONT UP" : Bool;
      "HIPOT & THICKNESS STAGE LIFT FRONT DOWN" : Bool;
      "HIPOT & THICKNESS STAGE LIFT REAR UP" : Bool;
      "HIPOT & THICKNESS STAGE LIFT REAR DOWN" : Bool;
      SPARE_4 : Bool;
      SPARE_5 : Bool;
   END_VAR
BEGIN
END_DATA_BLOCK

DATA_BLOCK "PM9"   // DB283
// stored: MemoryReserve 100
   VAR
      "FINAL VISION STAGE LIFT UP" : Bool;
      "FINAL VISION STAGE LIFT DOWN" : Bool;
      "FINAL VISION LIGHT UP" : Bool;
      "FINAL VISION LIGHT DOWN" : Bool;
      "LASER MARKING COVER UP" : Bool;
      "LASER MARKING COVER DOWN" : Bool;
      "LASER MARKING STAGE LIFT UP" : Bool;
      "LASER MARKING STAGE LIFT DOWN" : Bool;
      SPARE : Bool;
      SPARE_1 : Bool;
      "INS TRANSFER P&P CLAMP #1 CLOSE" : Bool;
      "INS TRANSFER P&P CLAMP #1 OPEN" : Bool;
      "INS TRANSFER P&P CLAMP #2 CLOSE" : Bool;
      "INS TRANSFER P&P CLAMP #2 OPEN" : Bool;
      "JR Unloading P&P CLAMP CLOSE" : Bool;
      "JR Unloading P&P CLAMP OPEN" : Bool;
   END_VAR
BEGIN
END_DATA_BLOCK

